KUKA KRL program: EPS_2_251825_SA34_A_20260116064118.src

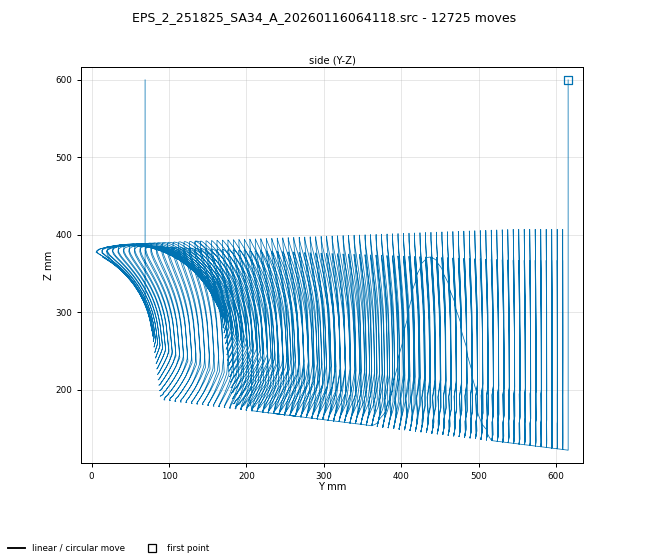
[picture p0: tool path of EPS_2_251825_SA34_A_20260116064118.src, 12725 of 12727 moves have a stored position in this frame; points joined in program order, loops and branches not executed]
&ACCESS RVP
&REL 4
&COMMENT QRS 19112012
&PARAM EDITMASK = *
DEF PART()
EXT BAS (BAS_COMMAND :IN,REAL :IN )
INT I
BAS (#INITMOV,0 )

;KUKA QRS Post kuka4.cps  Date:22-06-2017 !

File_ID=2990

QRS_PRE_INIT()

;Init var - Until changes are made in qrs_pre_init
Outlet_Square_prg=0
Inlet_1_Square_prg=0
Inlet_2_Square_prg=0
Inlet_3_Square_prg=0
Inlet_4_Square_prg=0
Inlet_5_Square_prg=0

Outlet_1={X 0.000, Y 546.330, Z 306.500, B 0.000, E1 0.000 }
Inlet_1={X 0.000, Y 549.180, Z 266.500, B 0.000, E1 160.000 }
Outlet_1_type=201
Inlet_1_type=201
;QRS#1=Sidecore dimensions
;QRS#2=200-8" PVC SDR 35
;QRS#3=200-8" PVC SDR 35
;QRS#4=
;QRS#5=
;QRS#6=
;QRS#7=
;QRS#8=
;QRS#9=12-08 PSX
;QRS#10=12-08 PSX
;QRS#11=
;QRS#12=
;QRS#13=
;QRS#14=
;QRS#15=
;QRS#16=1220x127x686 2,25'
;QRS#17=EPS Height
;QRS#18=407
;QRS#19=*
;QRS#20= UPDATED VERSION 22-06-2017
;QRS#21=*
Outlet_Square=0100
Inlet_1_Square=0100
Inlet_2_Square=0
Inlet_3_Square=0
Inlet_4_Square=0
Inlet_5_Square=0
Mill_Square=1
Outlet_Square_Prg=204
Inlet_1_Square_prg=204

QRS_INIT()

$ADVANCE=5

; T1
PTP {E1 173.645,E2 173.645}
PTP {X 0,Y 615.452,A -85,B 0,C 180,E1 173.645,E2 173.645,E3 0,E4 0,E5 0,E6 0}
QRS_SPEED_INIT()
LIN {X 0,Y 615.452,Z 600,A -85,B 0,C 180,E1 173.645,E2 173.645,E3 0,E4 0,E5 0,E6 0} C_VEL
LIN {X 0,Y 615.452,Z 131.871,A -85,B 0,C 180,E1 173.645,E2 173.645} C_VEL
LIN {X 0,Y 615.452,Z 123.693,A -85,B 0,C 180,E1 173.645,E2 173.645} C_VEL
LIN {X 0,Y 615.446,Z 121.693,A -85,B 0,C 180,E1 173.459,E2 173.459} C_VEL
LIN {X 0,Y 615.481,Z 121.699,A -85,B 0,C 180,E1 170.802,E2 170.802} C_VEL
LIN {X 0,Y 615.48,Z 121.688,A -85,B 0,C 180,E1 168.139,E2 168.139} C_VEL
LIN {X 0,Y 615.452,Z 121.694,A -85,B 0,C 180,E1 165.45,E2 165.45} C_VEL
LIN {X 0,Y 615.493,Z 121.695,A -85,B 0,C 180,E1 162.73,E2 162.73} C_VEL
LIN {X 0,Y 615.459,Z 121.69,A -85,B 0,C 180,E1 159.967,E2 159.967} C_VEL
LIN {X 0,Y 615.457,Z 121.693,A -85,B 0,C 180,E1 157.662,E2 157.662} C_VEL
LIN {X 0,Y 615.494,Z 121.696,A -85,B 0,C 180,E1 155.009,E2 155.009} C_VEL
LIN {X 0,Y 615.461,Z 121.69,A -85,B 0,C 180,E1 152.084,E2 152.084} C_VEL
LIN {X 0,Y 615.46,Z 121.694,A -85,B 0,C 180,E1 149.839,E2 149.839} C_VEL
LIN {X 0,Y 615.481,Z 121.699,A -85,B 0,C 180,E1 147.543,E2 147.543} C_VEL
LIN {X 0,Y 615.489,Z 121.693,A -85,B 0,C 180,E1 145.186,E2 145.186} C_VEL
LIN {X 0,Y 615.491,Z 121.683,A -85,B 0,C 180,E1 142.759,E2 142.759} C_VEL
LIN {X 0,Y 615.475,Z 121.697,A -85,B 0,C 180,E1 139.913,E2 139.913} C_VEL
LIN {X 0,Y 615.488,Z 121.684,A -85,B 0,C 180,E1 136.953,E2 136.953} C_VEL
LIN {X 0,Y 615.475,Z 121.695,A -85,B 0,C 180,E1 134.151,E2 134.151} C_VEL
LIN {X 0,Y 615.484,Z 121.69,A -85,B 0,C 180,E1 131.474,E2 131.474} C_VEL
LIN {X 0,Y 615.473,Z 121.689,A -85,B 0,C 180,E1 128.643,E2 128.643} C_VEL
LIN {X 0,Y 615.494,Z 136.384,A -85,B 0,C 180,E1 126.128,E2 126.128} C_VEL
LIN {X 0,Y 615.488,Z 153.64,A -85,B 0,C 180,E1 123.236,E2 123.236} C_VEL
LIN {X 0,Y 615.488,Z 156.2,A -85,B 0,C 180,E1 122.81,E2 122.81} C_VEL
LIN {X 0,Y 615.474,Z 263.278,A -85,B 0,C 180,E1 121.536,E2 121.536} C_VEL
LIN {X 0,Y 615.497,Z 276.678,A -85,B 0,C 180,E1 121.236,E2 121.236} C_VEL
LIN {X 0,Y 615.493,Z 289.09,A -85,B 0,C 180,E1 120.824,E2 120.824} C_VEL
LIN {X 0,Y 615.469,Z 299.786,A -85,B 0,C 180,E1 120.351,E2 120.351} C_VEL
LIN {X 0,Y 615.47,Z 311.326,A -85,B 0,C 180,E1 119.695,E2 119.695} C_VEL
LIN {X 0,Y 615.499,Z 321.929,A -85,B 0,C 180,E1 118.938,E2 118.938} C_VEL
LIN {X 0,Y 615.497,Z 330.569,A -85,B 0,C 180,E1 118.184,E2 118.184} C_VEL
LIN {X 0,Y 615.498,Z 338.385,A -85,B 0,C 180,E1 117.361,E2 117.361} C_VEL
LIN {X 0,Y 615.494,Z 345.548,A -85,B 0,C 180,E1 116.444,E2 116.444} C_VEL
LIN {X 0,Y 615.495,Z 352.739,A -85,B 0,C 180,E1 115.281,E2 115.281} C_VEL
LIN {X 0,Y 615.496,Z 357.591,A -85,B 0,C 180,E1 114.272,E2 114.272} C_VEL
LIN {X 0,Y 615.495,Z 361.489,A -85,B 0,C 180,E1 113.2,E2 113.2} C_VEL
LIN {X 0,Y 615.497,Z 364.191,A -85,B 0,C 180,E1 112.136,E2 112.136} C_VEL
LIN {X 0,Y 615.498,Z 365.382,A -85,B 0,C 180,E1 111.432,E2 111.432} C_VEL
LIN {X 0,Y 615.495,Z 366.208,A -85,B 0,C 180,E1 110.56,E2 110.56} C_VEL
LIN {X 0,Y 615.496,Z 366.2,A -85,B 0,C 180,E1 109.338,E2 109.338} C_VEL
LIN {X 0,Y 615.495,Z 365.535,A -85,B 0,C 180,E1 108.608,E2 108.608} C_VEL
LIN {X 0,Y 615.497,Z 364.55,A -85,B 0,C 180,E1 107.957,E2 107.957} C_VEL
LIN {X 0,Y 615.495,Z 363.056,A -85,B 0,C 180,E1 107.27,E2 107.27} C_VEL
LIN {X 0,Y 615.495,Z 360.608,A -85,B 0,C 180,E1 106.435,E2 106.435} C_VEL
LIN {X 0,Y 615.497,Z 355.768,A -85,B 0,C 180,E1 105.226,E2 105.226} C_VEL
LIN {X 0,Y 615.495,Z 350.565,A -85,B 0,C 180,E1 104.244,E2 104.244} C_VEL
LIN {X 0,Y 615.497,Z 343.595,A -85,B 0,C 180,E1 103.201,E2 103.201} C_VEL
LIN {X 0,Y 615.497,Z 335.207,A -85,B 0,C 180,E1 102.195,E2 102.195} C_VEL
LIN {X 0,Y 615.499,Z 326.571,A -85,B 0,C 180,E1 101.36,E2 101.36} C_VEL
LIN {X 0,Y 615.494,Z 315.975,A -85,B 0,C 180,E1 100.527,E2 100.527} C_VEL
LIN {X 0,Y 615.495,Z 305.473,A -85,B 0,C 180,E1 99.862,E2 99.862} C_VEL
LIN {X 0,Y 615.497,Z 293.798,A -85,B 0,C 180,E1 99.281,E2 99.281} C_VEL
LIN {X 0,Y 615.462,Z 281.785,A -85,B 0,C 180,E1 98.826,E2 98.826} C_VEL
LIN {X 0,Y 615.454,Z 269.574,A -85,B 0,C 180,E1 98.496,E2 98.496} C_VEL
LIN {X 0,Y 615.459,Z 257.497,A -85,B 0,C 180,E1 98.289,E2 98.289} C_VEL
LIN {X 0,Y 615.464,Z 156.157,A -85,B 0,C 180,E1 97.092,E2 97.092} C_VEL
LIN {X 0,Y 615.44,Z 141.171,A -85,B 0,C 180,E1 94.585,E2 94.585} C_VEL
LIN {X 0,Y 615.499,Z 125.645,A -85,B 0,C 180,E1 91.963,E2 91.963} C_VEL
LIN {X 0,Y 615.429,Z 121.699,A -85,B 0,C 180,E1 91.268,E2 91.268} C_VEL
LIN {X 0,Y 615.43,Z 121.699,A -85,B 0,C 180,E1 89.346,E2 89.346} C_VEL
LIN {X 0,Y 615.429,Z 121.699,A -85,B 0,C 180,E1 87.382,E2 87.382} C_VEL
LIN {X 0,Y 615.427,Z 121.699,A -85,B 0,C 180,E1 85.415,E2 85.415} C_VEL
LIN {X 0,Y 615.427,Z 121.699,A -85,B 0,C 180,E1 83.443,E2 83.443} C_VEL
LIN {X 0,Y 615.425,Z 121.699,A -85,B 0,C 180,E1 81.462,E2 81.462} C_VEL
LIN {X 0,Y 615.416,Z 121.699,A -85,B 0,C 180,E1 79.144,E2 79.144} C_VEL
LIN {X 0,Y 615.435,Z 121.699,A -85,B 0,C 180,E1 76.797,E2 76.797} C_VEL
LIN {X 0,Y 615.466,Z 121.7,A -85,B 0,C 180,E1 74.094,E2 74.094} C_VEL
LIN {X 0,Y 615.414,Z 121.699,A -85,B 0,C 180,E1 71.351,E2 71.351} C_VEL
LIN {X 0,Y 615.485,Z 121.699,A -85,B 0,C 180,E1 68.568,E2 68.568} C_VEL
LIN {X 0,Y 615.416,Z 121.7,A -85,B 0,C 180,E1 65.725,E2 65.725} C_VEL
LIN {X 0,Y 615.41,Z 121.7,A -85,B 0,C 180,E1 63.552,E2 63.552} C_VEL
LIN {X 0,Y 615.477,Z 121.703,A -85,B 0,C 180,E1 60.593,E2 60.593} C_VEL
LIN {X 0,Y 615.445,Z 121.7,A -85,B 0,C 180,E1 58.312,E2 58.312} C_VEL
LIN {X 0,Y 615.416,Z 121.7,A -85,B 0,C 180,E1 55.973,E2 55.973} C_VEL
LIN {X 0,Y 615.464,Z 121.7,A -85,B 0,C 180,E1 53.066,E2 53.066} C_VEL
LIN {X 0,Y 615.422,Z 121.7,A -85,B 0,C 180,E1 50.244,E2 50.244} C_VEL
LIN {X 0,Y 615.414,Z 121.699,A -85,B 0,C 180,E1 47.927,E2 47.927} C_VEL
LIN {X 0,Y 615.416,Z 121.7,A -85,B 0,C 180,E1 45.843,E2 45.843} C_VEL
LIN {X 0,Y 615.475,Z 121.7,A -85,B 0,C 180,E1 43.245,E2 43.245} C_VEL
LIN {X 0,Y 615.437,Z 121.698,A -85,B 0,C 180,E1 40.61,E2 40.61} C_VEL
LIN {X 0,Y 615.466,Z 121.698,A -85,B 0,C 180,E1 38.905,E2 38.905} C_VEL
LIN {X 0,Y 615.421,Z 121.699,A -85,B 0,C 180,E1 36.429,E2 36.429} C_VEL
LIN {X 0,Y 615.469,Z 121.7,A -85,B 0,C 180,E1 33.531,E2 33.531} C_VEL
LIN {X 0,Y 615.447,Z 121.698,A -85,B 0,C 180,E1 30.921,E2 30.921} C_VEL
LIN {X 0,Y 615.419,Z 121.698,A -85,B 0,C 180,E1 28.437,E2 28.437} C_VEL
LIN {X 0,Y 615.471,Z 121.7,A -85,B 0,C 180,E1 25.716,E2 25.716} C_VEL
LIN {X 0,Y 615.428,Z 121.697,A -85,B 0,C 180,E1 22.846,E2 22.846} C_VEL
LIN {X 0,Y 615.421,Z 121.698,A -85,B 0,C 180,E1 20.539,E2 20.539} C_VEL
LIN {X 0,Y 615.465,Z 121.699,A -85,B 0,C 180,E1 17.957,E2 17.957} C_VEL
LIN {X 0,Y 615.445,Z 121.696,A -85,B 0,C 180,E1 15.227,E2 15.227} C_VEL
LIN {X 0,Y 615.439,Z 121.697,A -85,B 0,C 180,E1 13.202,E2 13.202} C_VEL
LIN {X 0,Y 615.423,Z 121.697,A -85,B 0,C 180,E1 10.854,E2 10.854} C_VEL
LIN {X 0,Y 615.434,Z 121.698,A -85,B 0,C 180,E1 8.537,E2 8.537} C_VEL
LIN {X 0,Y 615.499,Z 121.696,A -85,B 0,C 180,E1 5.898,E2 5.898} C_VEL
LIN {X 0,Y 615.431,Z 121.696,A -85,B 0,C 180,E1 3.273,E2 3.273} C_VEL
LIN {X 0,Y 615.429,Z 121.697,A -85,B 0,C 180,E1 1.308,E2 1.308} C_VEL
LIN {X 0,Y 615.431,Z 121.696,A -85,B 0,C 180,E1 -0.655,E2 -0.655} C_VEL
LIN {X 0,Y 615.429,Z 121.697,A -85,B 0,C 180,E1 -2.618,E2 -2.618} C_VEL
LIN {X 0,Y 615.431,Z 121.696,A -85,B 0,C 180,E1 -4.585,E2 -4.585} C_VEL
LIN {X 0,Y 615.431,Z 121.696,A -85,B 0,C 180,E1 -6.558,E2 -6.558} C_VEL
LIN {X 0,Y 615.43,Z 121.696,A -85,B 0,C 180,E1 -8.538,E2 -8.538} C_VEL
LIN {X 0,Y 615.431,Z 121.697,A -85,B 0,C 180,E1 -10.858,E2 -10.858} C_VEL
LIN {X 0,Y 615.456,Z 121.7,A -85,B 0,C 180,E1 -13.202,E2 -13.202} C_VEL
LIN {X 0,Y 615.465,Z 121.694,A -85,B 0,C 180,E1 -15.906,E2 -15.906} C_VEL
LIN {X 0,Y 615.454,Z 121.694,A -85,B 0,C 180,E1 -17.958,E2 -17.958} C_VEL
LIN {X 0,Y 615.431,Z 121.697,A -85,B 0,C 180,E1 -20.541,E2 -20.541} C_VEL
LIN {X 0,Y 615.45,Z 121.698,A -85,B 0,C 180,E1 -22.846,E2 -22.846} C_VEL
LIN {X 0,Y 615.463,Z 121.693,A -85,B 0,C 180,E1 -25.717,E2 -25.717} C_VEL
LIN {X 0,Y 615.441,Z 121.694,A -85,B 0,C 180,E1 -27.918,E2 -27.918} C_VEL
LIN {X 0,Y 615.432,Z 121.695,A -85,B 0,C 180,E1 -30.163,E2 -30.163} C_VEL
LIN {X 0,Y 615.441,Z 121.697,A -85,B 0,C 180,E1 -32.461,E2 -32.461} C_VEL
LIN {X 0,Y 615.478,Z 121.7,A -85,B 0,C 180,E1 -34.816,E2 -34.816} C_VEL
LIN {X 0,Y 615.487,Z 121.692,A -85,B 0,C 180,E1 -37.243,E2 -37.243} C_VEL
LIN {X 0,Y 615.436,Z 121.695,A -85,B 0,C 180,E1 -39.754,E2 -39.754} C_VEL
LIN {X 0,Y 615.434,Z 121.697,A -85,B 0,C 180,E1 -42.074,E2 -42.074} C_VEL
LIN {X 0,Y 615.442,Z 121.697,A -85,B 0,C 180,E1 -44.154,E2 -44.154} C_VEL
LIN {X 0,Y 615.488,Z 121.693,A -85,B 0,C 180,E1 -46.953,E2 -46.953} C_VEL
LIN {X 0,Y 615.448,Z 121.693,A -85,B 0,C 180,E1 -49.39,E2 -49.39} C_VEL
LIN {X 0,Y 615.445,Z 121.697,A -85,B 0,C 180,E1 -51.994,E2 -51.994} C_VEL
LIN {X 0,Y 615.487,Z 121.699,A -85,B 0,C 180,E1 -54.384,E2 -54.384} C_VEL
LIN {X 0,Y 615.486,Z 121.692,A -85,B 0,C 180,E1 -56.763,E2 -56.763} C_VEL
LIN {X 0,Y 615.456,Z 121.692,A -85,B 0,C 180,E1 -59.078,E2 -59.078} C_VEL
LIN {X 0,Y 615.439,Z 121.695,A -85,B 0,C 180,E1 -61.559,E2 -61.559} C_VEL
LIN {X 0,Y 615.494,Z 121.694,A -85,B 0,C 180,E1 -64.431,E2 -64.431} C_VEL
LIN {X 0,Y 615.442,Z 121.693,A -85,B 0,C 180,E1 -67.153,E2 -67.153} C_VEL
LIN {X 0,Y 615.441,Z 121.787,A -85,B 0,C 180,E1 -67.44,E2 -67.44} C_VEL
LIN {X 0,Y 615.478,Z 140.396,A -85,B 0,C 180,E1 -69.967,E2 -69.967} C_VEL
LIN {X 0,Y 615.47,Z 161.075,A -85,B 0,C 180,E1 -72.729,E2 -72.729} C_VEL
LIN {X 0,Y 615.472,Z 181.731,A -85,B 0,C 180,E1 -75.45,E2 -75.45} C_VEL
LIN {X 0,Y 615.454,Z 194.469,A -85,B 0,C 180,E1 -77.113,E2 -77.113} C_VEL
LIN {X 0,Y 615.488,Z 302.818,A -85,B 0,C 180,E1 -78.41,E2 -78.41} C_VEL
LIN {X 0,Y 615.477,Z 315.338,A -85,B 0,C 180,E1 -78.681,E2 -78.681} C_VEL
LIN {X 0,Y 615.488,Z 328.619,A -85,B 0,C 180,E1 -79.113,E2 -79.113} C_VEL
LIN {X 0,Y 615.477,Z 340.475,A -85,B 0,C 180,E1 -79.639,E2 -79.639} C_VEL
LIN {X 0,Y 615.494,Z 351.991,A -85,B 0,C 180,E1 -80.304,E2 -80.304} C_VEL
LIN {X 0,Y 615.499,Z 362.339,A -85,B 0,C 180,E1 -81.05,E2 -81.05} C_VEL
LIN {X 0,Y 615.497,Z 370.81,A -85,B 0,C 180,E1 -81.794,E2 -81.794} C_VEL
LIN {X 0,Y 615.498,Z 378.605,A -85,B 0,C 180,E1 -82.619,E2 -82.619} C_VEL
LIN {X 0,Y 615.496,Z 386.202,A -85,B 0,C 180,E1 -83.608,E2 -83.608} C_VEL
LIN {X 0,Y 615.498,Z 393.204,A -85,B 0,C 180,E1 -84.759,E2 -84.759} C_VEL
LIN {X 0,Y 615.494,Z 397.851,A -85,B 0,C 180,E1 -85.743,E2 -85.743} C_VEL
LIN {X 0,Y 615.494,Z 401.398,A -85,B 0,C 180,E1 -86.727,E2 -86.727} C_VEL
LIN {X 0,Y 615.497,Z 403.233,A -85,B 0,C 180,E1 -87.382,E2 -87.382} C_VEL
LIN {X 0,Y 615.5,Z 404.607,A -85,B 0,C 180,E1 -88.037,E2 -88.037} C_VEL
LIN {X 0,Y 615.496,Z 406.173,A -85,B 0,C 180,E1 -89.346,E2 -89.346} C_VEL
LIN {X 0,Y 615.494,Z 406.389,A -85,B 0,C 180,E1 -90,E2 -90} C_VEL
LIN {X 0,Y 615.495,Z 405.58,A -85,B 0,C 180,E1 -91.308,E2 -91.308} C_VEL
LIN {X 0,Y 615.5,Z 404.608,A -85,B 0,C 180,E1 -91.963,E2 -91.963} C_VEL
LIN {X 0,Y 615.497,Z 403.233,A -85,B 0,C 180,E1 -92.618,E2 -92.618} C_VEL
LIN {X 0,Y 615.496,Z 400.35,A -85,B 0,C 180,E1 -93.601,E2 -93.601} C_VEL
LIN {X 0,Y 615.498,Z 396.442,A -85,B 0,C 180,E1 -94.584,E2 -94.584} C_VEL
LIN {X 0,Y 615.499,Z 391.405,A -85,B 0,C 180,E1 -95.57,E2 -95.57} C_VEL
LIN {X 0,Y 615.497,Z 384.87,A -85,B 0,C 180,E1 -96.583,E2 -96.583} C_VEL
LIN {X 0,Y 615.497,Z 377.134,A -85,B 0,C 180,E1 -97.545,E2 -97.545} C_VEL
LIN {X 0,Y 615.498,Z 369.045,A -85,B 0,C 180,E1 -98.371,E2 -98.371} C_VEL
LIN {X 0,Y 615.499,Z 359.168,A -85,B 0,C 180,E1 -99.199,E2 -99.199} C_VEL
LIN {X 0,Y 615.488,Z 347.982,A -85,B 0,C 180,E1 -99.945,E2 -99.945} C_VEL
LIN {X 0,Y 615.482,Z 337.024,A -85,B 0,C 180,E1 -100.527,E2 -100.527} C_VEL
LIN {X 0,Y 615.48,Z 324.491,A -85,B 0,C 180,E1 -101.04,E2 -101.04} C_VEL
LIN {X 0,Y 615.479,Z 312.068,A -85,B 0,C 180,E1 -101.402,E2 -101.402} C_VEL
LIN {X 0,Y 615.493,Z 298.466,A -85,B 0,C 180,E1 -101.652,E2 -101.652} C_VEL
LIN {X 0,Y 615.454,Z 194.471,A -85,B 0,C 180,E1 -102.887,E2 -102.887} C_VEL
LIN {X 0,Y 615.496,Z 172.696,A -85,B 0,C 180,E1 -105.735,E2 -105.735} C_VEL
LIN {X 0,Y 615.455,Z 152.319,A -85,B 0,C 180,E1 -108.436,E2 -108.436} C_VEL
LIN {X 0,Y 615.475,Z 132.637,A -85,B 0,C 180,E1 -111.081,E2 -111.081} C_VEL
LIN {X 0,Y 615.44,Z 121.695,A -85,B 0,C 180,E1 -112.592,E2 -112.592} C_VEL
LIN {X 0,Y 615.451,Z 121.692,A -85,B 0,C 180,E1 -114.993,E2 -114.993} C_VEL
LIN {X 0,Y 615.468,Z 121.699,A -85,B 0,C 180,E1 -117.916,E2 -117.916} C_VEL
LIN {X 0,Y 615.442,Z 121.697,A -85,B 0,C 180,E1 -120.163,E2 -120.163} C_VEL
LIN {X 0,Y 615.432,Z 121.696,A -85,B 0,C 180,E1 -122.461,E2 -122.461} C_VEL
LIN {X 0,Y 615.451,Z 121.694,A -85,B 0,C 180,E1 -124.818,E2 -124.818} C_VEL
LIN {X 0,Y 615.495,Z 121.697,A -85,B 0,C 180,E1 -127.242,E2 -127.242} C_VEL
LIN {X 0,Y 615.444,Z 121.699,A -85,B 0,C 180,E1 -129.754,E2 -129.754} C_VEL
LIN {X 0,Y 615.425,Z 121.698,A -85,B 0,C 180,E1 -132.073,E2 -132.073} C_VEL
LIN {X 0,Y 615.423,Z 121.698,A -85,B 0,C 180,E1 -134.156,E2 -134.156} C_VEL
LIN {X 0,Y 615.469,Z 121.697,A -85,B 0,C 180,E1 -136.753,E2 -136.753} C_VEL
LIN {X 0,Y 615.444,Z 121.7,A -85,B 0,C 180,E1 -139.39,E2 -139.39} C_VEL
LIN {X 0,Y 615.473,Z 121.7,A -85,B 0,C 180,E1 -141.094,E2 -141.094} C_VEL
LIN {X 0,Y 615.418,Z 121.7,A -85,B 0,C 180,E1 -143.57,E2 -143.57} C_VEL
LIN {X 0,Y 615.46,Z 121.7,A -85,B 0,C 180,E1 -146.47,E2 -146.47} C_VEL
LIN {X 0,Y 615.446,Z 121.699,A -85,B 0,C 180,E1 -149.078,E2 -149.078} C_VEL
LIN {X 0,Y 615.417,Z 121.699,A -85,B 0,C 180,E1 -151.562,E2 -151.562} C_VEL
LIN {X 0,Y 615.47,Z 121.7,A -85,B 0,C 180,E1 -154.283,E2 -154.283} C_VEL
LIN {X 0,Y 615.43,Z 121.697,A -85,B 0,C 180,E1 -157.153,E2 -157.153} C_VEL
LIN {X 0,Y 615.424,Z 121.698,A -85,B 0,C 180,E1 -159.46,E2 -159.46} C_VEL
LIN {X 0,Y 615.473,Z 121.699,A -85,B 0,C 180,E1 -162.042,E2 -162.042} C_VEL
LIN {X 0,Y 615.448,Z 121.695,A -85,B 0,C 180,E1 -164.773,E2 -164.773} C_VEL
LIN {X 0,Y 615.443,Z 121.695,A -85,B 0,C 180,E1 -166.797,E2 -166.797} C_VEL
LIN {X 0,Y 615.432,Z 121.696,A -85,B 0,C 180,E1 -169.141,E2 -169.141} C_VEL
LIN {X 0,Y 615.448,Z 121.698,A -85,B 0,C 180,E1 -171.462,E2 -171.462} C_VEL
LIN {X 0,Y 615.499,Z 121.691,A -85,B 0,C 180,E1 -174.101,E2 -174.101} C_VEL
LIN {X 0,Y 615.44,Z 121.694,A -85,B 0,C 180,E1 -176.726,E2 -176.726} C_VEL
LIN {X 0,Y 615.441,Z 121.694,A -85,B 0,C 180,E1 -178.691,E2 -178.691} C_VEL
LIN {X 0,Y 615.465,Z 121.698,A -85,B 0,C 180,E1 -181.308,E2 -181.308} C_VEL
LIN {X 0,Y 615.486,Z 121.691,A -85,B 0,C 180,E1 -183.928,E2 -183.928} C_VEL
LIN {X 0,Y 615.446,Z 121.693,A -85,B 0,C 180,E1 -186.541,E2 -186.541} C_VEL
LIN {X 0,Y 614.789,Z 121.846,A -85,B 0,C 180,E1 -187.087,E2 -187.087} C_VEL
LIN {X 0,Y 611.974,Z 122.251,A -85,B 0,C 180,E1 -187.974,E2 -187.974} C_VEL
LIN {X 0,Y 609.586,Z 122.567,A -85,B 0,C 180,E1 -188.686,E2 -188.686} C_VEL
LIN {X 0,Y 608.549,Z 122.687,A -85,B 0,C 180,E1 -189.236,E2 -189.236} C_VEL
LIN {X 0,Y 608.459,Z 122.695,A -85,B 0,C 180,E1 -189.422,E2 -189.422} C_VEL
LIN {X 0,Y 608.451,Z 122.689,A -85,B 0,C 180,E1 -192,E2 -192} C_VEL
LIN {X 0,Y 608.449,Z 122.688,A -85,B 0,C 180,E1 -194.038,E2 -194.038} C_VEL
LIN {X 0,Y 608.45,Z 122.69,A -85,B 0,C 180,E1 -196.522,E2 -196.522} C_VEL
LIN {X 0,Y 608.448,Z 122.69,A -85,B 0,C 180,E1 -199.57,E2 -199.57} C_VEL
LIN {X 0,Y 608.434,Z 122.692,A -85,B 0,C 180,E1 -202.406,E2 -202.406} C_VEL
LIN {X 0,Y 608.453,Z 122.691,A -85,B 0,C 180,E1 -205.3,E2 -205.3} C_VEL
LIN {X 0,Y 608.442,Z 122.69,A -85,B 0,C 180,E1 -207.518,E2 -207.518} C_VEL
LIN {X 0,Y 608.446,Z 122.689,A -85,B 0,C 180,E1 -209.967,E2 -209.967} C_VEL
LIN {X 0,Y 608.457,Z 122.693,A -85,B 0,C 180,E1 -212.879,E2 -212.879} C_VEL
LIN {X 0,Y 608.435,Z 122.691,A -85,B 0,C 180,E1 -215.278,E2 -215.278} C_VEL
LIN {X 0,Y 608.461,Z 122.688,A -85,B 0,C 180,E1 -217.746,E2 -217.746} C_VEL
LIN {X 0,Y 608.447,Z 122.699,A -85,B 0,C 180,E1 -220.328,E2 -220.328} C_VEL
LIN {X 0,Y 608.456,Z 122.688,A -85,B 0,C 180,E1 -222.959,E2 -222.959} C_VEL
LIN {X 0,Y 608.447,Z 122.692,A -85,B 0,C 180,E1 -225.736,E2 -225.736} C_VEL
LIN {X 0,Y 608.462,Z 122.689,A -85,B 0,C 180,E1 -228.657,E2 -228.657} C_VEL
LIN {X 0,Y 608.462,Z 122.787,A -85,B 0,C 180,E1 -231.332,E2 -231.332} C_VEL
LIN {X 0,Y 608.479,Z 138.082,A -85,B 0,C 180,E1 -233.95,E2 -233.95} C_VEL
LIN {X 0,Y 608.46,Z 154.529,A -85,B 0,C 180,E1 -236.726,E2 -236.726} C_VEL
LIN {X 0,Y 608.473,Z 156.462,A -85,B 0,C 180,E1 -237.044,E2 -237.044} C_VEL
LIN {X 0,Y 608.534,Z 263.716,A -85,B 0,C 180,E1 -238.336,E2 -238.336} C_VEL
LIN {X 0,Y 608.534,Z 277.004,A -85,B 0,C 180,E1 -238.639,E2 -238.639} C_VEL
LIN {X 0,Y 608.526,Z 289.836,A -85,B 0,C 180,E1 -239.073,E2 -239.073} C_VEL
LIN {X 0,Y 608.486,Z 301.644,A -85,B 0,C 180,E1 -239.618,E2 -239.618} C_VEL
LIN {X 0,Y 608.463,Z 313.409,A -85,B 0,C 180,E1 -240.315,E2 -240.315} C_VEL
LIN {X 0,Y 608.488,Z 323.927,A -85,B 0,C 180,E1 -241.098,E2 -241.098} C_VEL
LIN {X 0,Y 608.485,Z 332.9,A -85,B 0,C 180,E1 -241.923,E2 -241.923} C_VEL
LIN {X 0,Y 608.462,Z 341.754,A -85,B 0,C 180,E1 -242.92,E2 -242.92} C_VEL
LIN {X 0,Y 608.434,Z 349.174,A -85,B 0,C 180,E1 -243.964,E2 -243.964} C_VEL
LIN {X 0,Y 608.43,Z 355.309,A -85,B 0,C 180,E1 -245.063,E2 -245.063} C_VEL
LIN {X 0,Y 608.441,Z 359.985,A -85,B 0,C 180,E1 -246.154,E2 -246.154} C_VEL
LIN {X 0,Y 608.44,Z 362.405,A -85,B 0,C 180,E1 -246.876,E2 -246.876} C_VEL
LIN {X 0,Y 608.429,Z 364.248,A -85,B 0,C 180,E1 -247.593,E2 -247.593} C_VEL
LIN {X 0,Y 608.419,Z 365.612,A -85,B 0,C 180,E1 -248.307,E2 -248.307} C_VEL
LIN {X 0,Y 608.44,Z 366.744,A -85,B 0,C 180,E1 -249.327,E2 -249.327} C_VEL
LIN {X 0,Y 608.416,Z 366.916,A -85,B 0,C 180,E1 -250.428,E2 -250.428} C_VEL
LIN {X 0,Y 608.426,Z 366.271,A -85,B 0,C 180,E1 -251.295,E2 -251.295} C_VEL
LIN {X 0,Y 608.419,Z 364.193,A -85,B 0,C 180,E1 -252.522,E2 -252.522} C_VEL
LIN {X 0,Y 608.426,Z 361.552,A -85,B 0,C 180,E1 -253.483,E2 -253.483} C_VEL
LIN {X 0,Y 608.43,Z 357.335,A -85,B 0,C 180,E1 -254.593,E2 -254.593} C_VEL
LIN {X 0,Y 608.434,Z 352.189,A -85,B 0,C 180,E1 -255.62,E2 -255.62} C_VEL
LIN {X 0,Y 608.445,Z 345.722,A -85,B 0,C 180,E1 -256.643,E2 -256.643} C_VEL
LIN {X 0,Y 608.46,Z 337.624,A -85,B 0,C 180,E1 -257.662,E2 -257.662} C_VEL
LIN {X 0,Y 608.469,Z 329.402,A -85,B 0,C 180,E1 -258.507,E2 -258.507} C_VEL
LIN {X 0,Y 608.5,Z 319.397,A -85,B 0,C 180,E1 -259.351,E2 -259.351} C_VEL
LIN {X 0,Y 608.492,Z 308.141,A -85,B 0,C 180,E1 -260.107,E2 -260.107} C_VEL
LIN {X 0,Y 608.51,Z 297.156,A -85,B 0,C 180,E1 -260.695,E2 -260.695} C_VEL
LIN {X 0,Y 608.511,Z 285.043,A -85,B 0,C 180,E1 -261.197,E2 -261.197} C_VEL
LIN {X 0,Y 608.521,Z 272.391,A -85,B 0,C 180,E1 -261.574,E2 -261.574} C_VEL
LIN {X 0,Y 608.511,Z 259.154,A -85,B 0,C 180,E1 -261.825,E2 -261.825} C_VEL
LIN {X 0,Y 608.45,Z 156.374,A -85,B 0,C 180,E1 -263.055,E2 -263.055} C_VEL
LIN {X 0,Y 608.441,Z 140.716,A -85,B 0,C 180,E1 -265.694,E2 -265.694} C_VEL
LIN {X 0,Y 608.444,Z 123.264,A -85,B 0,C 180,E1 -268.676,E2 -268.676} C_VEL
LIN {X 0,Y 608.413,Z 122.694,A -85,B 0,C 180,E1 -268.8,E2 -268.8} C_VEL
LIN {X 0,Y 608.408,Z 122.695,A -85,B 0,C 180,E1 -270.662,E2 -270.662} C_VEL
LIN {X 0,Y 608.425,Z 122.693,A -85,B 0,C 180,E1 -272.648,E2 -272.648} C_VEL
LIN {X 0,Y 608.413,Z 122.694,A -85,B 0,C 180,E1 -275.302,E2 -275.302} C_VEL
LIN {X 0,Y 608.464,Z 122.695,A -85,B 0,C 180,E1 -277.967,E2 -277.967} C_VEL
LIN {X 0,Y 608.402,Z 122.694,A -85,B 0,C 180,E1 -280.651,E2 -280.651} C_VEL
LIN {X 0,Y 608.425,Z 122.695,A -85,B 0,C 180,E1 -283.358,E2 -283.358} C_VEL
LIN {X 0,Y 608.425,Z 122.695,A -85,B 0,C 180,E1 -286.095,E2 -286.095} C_VEL
LIN {X 0,Y 608.396,Z 122.695,A -85,B 0,C 180,E1 -288.872,E2 -288.872} C_VEL
LIN {X 0,Y 608.447,Z 122.696,A -85,B 0,C 180,E1 -291.693,E2 -291.693} C_VEL
LIN {X 0,Y 608.402,Z 122.694,A -85,B 0,C 180,E1 -294.574,E2 -294.574} C_VEL
LIN {X 0,Y 608.456,Z 122.694,A -85,B 0,C 180,E1 -297.204,E2 -297.204} C_VEL
LIN {X 0,Y 608.4,Z 122.696,A -85,B 0,C 180,E1 -299.961,E2 -299.961} C_VEL
LIN {X 0,Y 608.402,Z 122.694,A -85,B 0,C 180,E1 -302.514,E2 -302.514} C_VEL
LIN {X 0,Y 608.406,Z 122.703,A -85,B 0,C 180,E1 -305.281,E2 -305.281} C_VEL
LIN {X 0,Y 608.423,Z 122.693,A -85,B 0,C 180,E1 -307.75,E2 -307.75} C_VEL
LIN {X 0,Y 608.4,Z 122.695,A -85,B 0,C 180,E1 -310.324,E2 -310.324} C_VEL
LIN {X 0,Y 608.439,Z 122.699,A -85,B 0,C 180,E1 -312.962,E2 -312.962} C_VEL
LIN {X 0,Y 608.4,Z 122.695,A -85,B 0,C 180,E1 -315.742,E2 -315.742} C_VEL
LIN {X 0,Y 608.401,Z 122.694,A -85,B 0,C 180,E1 -317.934,E2 -317.934} C_VEL
LIN {X 0,Y 608.433,Z 122.699,A -85,B 0,C 180,E1 -320.708,E2 -320.708} C_VEL
LIN {X 0,Y 608.432,Z 122.695,A -85,B 0,C 180,E1 -323.084,E2 -323.084} C_VEL
LIN {X 0,Y 608.42,Z 122.692,A -85,B 0,C 180,E1 -325.528,E2 -325.528} C_VEL
LIN {X 0,Y 608.416,Z 122.693,A -85,B 0,C 180,E1 -327.903,E2 -327.903} C_VEL
LIN {X 0,Y 608.435,Z 122.694,A -85,B 0,C 180,E1 -330.219,E2 -330.219} C_VEL
LIN {X 0,Y 608.398,Z 122.695,A -85,B 0,C 180,E1 -333.224,E2 -333.224} C_VEL
LIN {X 0,Y 608.409,Z 122.693,A -85,B 0,C 180,E1 -335.427,E2 -335.427} C_VEL
LIN {X 0,Y 608.451,Z 122.697,A -85,B 0,C 180,E1 -338.308,E2 -338.308} C_VEL
LIN {X 0,Y 608.411,Z 122.693,A -85,B 0,C 180,E1 -341.302,E2 -341.302} C_VEL
LIN {X 0,Y 608.432,Z 122.695,A -85,B 0,C 180,E1 -343.906,E2 -343.906} C_VEL
LIN {X 0,Y 608.432,Z 122.693,A -85,B 0,C 180,E1 -346.643,E2 -346.643} C_VEL
LIN {X 0,Y 608.41,Z 122.693,A -85,B 0,C 180,E1 -349.35,E2 -349.35} C_VEL
LIN {X 0,Y 608.472,Z 122.696,A -85,B 0,C 180,E1 -352.033,E2 -352.033} C_VEL
LIN {X 0,Y 608.418,Z 122.693,A -85,B 0,C 180,E1 -354.698,E2 -354.698} C_VEL
LIN {X 0,Y 608.434,Z 122.692,A -85,B 0,C 180,E1 -357.352,E2 -357.352} C_VEL
LIN {X 0,Y 608.478,Z 122.692,A -85,B 0,C 180,E1 -360,E2 -360} C_VEL
LIN {X 0,Y 608.426,Z 122.691,A -85,B 0,C 180,E1 -362.649,E2 -362.649} C_VEL
LIN {X 0,Y 608.431,Z 122.694,A -85,B 0,C 180,E1 -365.303,E2 -365.303} C_VEL
LIN {X 0,Y 608.469,Z 122.69,A -85,B 0,C 180,E1 -367.967,E2 -367.967} C_VEL
LIN {X 0,Y 608.432,Z 122.692,A -85,B 0,C 180,E1 -370.935,E2 -370.935} C_VEL
LIN {X 0,Y 608.44,Z 122.697,A -85,B 0,C 180,E1 -373.357,E2 -373.357} C_VEL
LIN {X 0,Y 608.429,Z 122.692,A -85,B 0,C 180,E1 -376.095,E2 -376.095} C_VEL
LIN {X 0,Y 608.436,Z 122.692,A -85,B 0,C 180,E1 -378.871,E2 -378.871} C_VEL
LIN {X 0,Y 608.458,Z 122.691,A -85,B 0,C 180,E1 -381.692,E2 -381.692} C_VEL
LIN {X 0,Y 608.422,Z 122.693,A -85,B 0,C 180,E1 -384.573,E2 -384.573} C_VEL
LIN {X 0,Y 608.482,Z 122.694,A -85,B 0,C 180,E1 -387.207,E2 -387.207} C_VEL
LIN {X 0,Y 608.412,Z 122.693,A -85,B 0,C 180,E1 -389.961,E2 -389.961} C_VEL
LIN {X 0,Y 608.425,Z 122.694,A -85,B 0,C 180,E1 -392.516,E2 -392.516} C_VEL
LIN {X 0,Y 608.423,Z 122.696,A -85,B 0,C 180,E1 -395.279,E2 -395.279} C_VEL
LIN {X 0,Y 608.437,Z 122.69,A -85,B 0,C 180,E1 -397.749,E2 -397.749} C_VEL
LIN {X 0,Y 608.438,Z 122.692,A -85,B 0,C 180,E1 -400.327,E2 -400.327} C_VEL
LIN {X 0,Y 608.461,Z 122.689,A -85,B 0,C 180,E1 -403.307,E2 -403.307} C_VEL
LIN {X 0,Y 608.435,Z 122.692,A -85,B 0,C 180,E1 -406.127,E2 -406.127} C_VEL
LIN {X 0,Y 608.457,Z 122.694,A -85,B 0,C 180,E1 -408.823,E2 -408.823} C_VEL
LIN {X 0,Y 608.416,Z 122.692,A -85,B 0,C 180,E1 -411.407,E2 -411.407} C_VEL
LIN {X 0,Y 608.437,Z 122.692,A -85,B 0,C 180,E1 -413.956,E2 -413.956} C_VEL
LIN {X 0,Y 608.45,Z 122.697,A -85,B 0,C 180,E1 -416.328,E2 -416.328} C_VEL
LIN {X 0,Y 608.446,Z 122.693,A -85,B 0,C 180,E1 -418.733,E2 -418.733} C_VEL
LIN {X 0,Y 608.434,Z 122.69,A -85,B 0,C 180,E1 -421.387,E2 -421.387} C_VEL
LIN {X 0,Y 608.432,Z 122.696,A -85,B 0,C 180,E1 -423.964,E2 -423.964} C_VEL
LIN {X 0,Y 608.43,Z 122.693,A -85,B 0,C 180,E1 -426.875,E2 -426.875} C_VEL
LIN {X 0,Y 608.435,Z 122.818,A -85,B 0,C 180,E1 -427.309,E2 -427.309} C_VEL
LIN {X 0,Y 608.573,Z 138.081,A -85,B 0,C 180,E1 -429.413,E2 -429.413} C_VEL
LIN {X 0,Y 608.533,Z 158.527,A -85,B 0,C 180,E1 -432.178,E2 -432.178} C_VEL
LIN {X 0,Y 608.493,Z 179.239,A -85,B 0,C 180,E1 -434.937,E2 -434.937} C_VEL
LIN {X 0,Y 608.441,Z 194.611,A -85,B 0,C 180,E1 -436.962,E2 -436.962} C_VEL
LIN {X 0,Y 608.569,Z 245.207,A -85,B 0,C 180,E1 -437.579,E2 -437.579} C_VEL
LIN {X 0,Y 608.547,Z 302.935,A -85,B 0,C 180,E1 -438.276,E2 -438.276} C_VEL
LIN {X 0,Y 608.512,Z 316.209,A -85,B 0,C 180,E1 -438.571,E2 -438.571} C_VEL
LIN {X 0,Y 608.514,Z 328.629,A -85,B 0,C 180,E1 -438.982,E2 -438.982} C_VEL
LIN {X 0,Y 608.499,Z 340.631,A -85,B 0,C 180,E1 -439.519,E2 -439.519} C_VEL
LIN {X 0,Y 608.484,Z 352.194,A -85,B 0,C 180,E1 -440.191,E2 -440.191} C_VEL
LIN {X 0,Y 608.485,Z 362.591,A -85,B 0,C 180,E1 -440.946,E2 -440.946} C_VEL
LIN {X 0,Y 608.475,Z 371.11,A -85,B 0,C 180,E1 -441.699,E2 -441.699} C_VEL
LIN {X 0,Y 608.471,Z 378.959,A -85,B 0,C 180,E1 -442.534,E2 -442.534} C_VEL
LIN {X 0,Y 608.461,Z 386.286,A -85,B 0,C 180,E1 -443.484,E2 -443.484} C_VEL
LIN {X 0,Y 608.451,Z 391.865,A -85,B 0,C 180,E1 -444.365,E2 -444.365} C_VEL
LIN {X 0,Y 608.432,Z 396.949,A -85,B 0,C 180,E1 -445.362,E2 -445.362} C_VEL
LIN {X 0,Y 608.449,Z 400.896,A -85,B 0,C 180,E1 -446.357,E2 -446.357} C_VEL
LIN {X 0,Y 608.425,Z 403.809,A -85,B 0,C 180,E1 -447.352,E2 -447.352} C_VEL
LIN {X 0,Y 608.445,Z 405.201,A -85,B 0,C 180,E1 -448.014,E2 -448.014} C_VEL
LIN {X 0,Y 608.438,Z 406.783,A -85,B 0,C 180,E1 -449.338,E2 -449.338} C_VEL
LIN {X 0,Y 608.434,Z 407,A -85,B 0,C 180,E1 -450,E2 -450} C_VEL
LIN {X 0,Y 608.448,Z 406.184,A -85,B 0,C 180,E1 -451.324,E2 -451.324} C_VEL
LIN {X 0,Y 608.445,Z 405.202,A -85,B 0,C 180,E1 -451.986,E2 -451.986} C_VEL
LIN {X 0,Y 608.425,Z 403.809,A -85,B 0,C 180,E1 -452.648,E2 -452.648} C_VEL
LIN {X 0,Y 608.449,Z 400.896,A -85,B 0,C 180,E1 -453.642,E2 -453.642} C_VEL
LIN {X 0,Y 608.432,Z 396.95,A -85,B 0,C 180,E1 -454.638,E2 -454.638} C_VEL
LIN {X 0,Y 608.438,Z 390.877,A -85,B 0,C 180,E1 -455.801,E2 -455.801} C_VEL
LIN {X 0,Y 608.462,Z 384.236,A -85,B 0,C 180,E1 -456.799,E2 -456.799} C_VEL
LIN {X 0,Y 608.456,Z 375.99,A -85,B 0,C 180,E1 -457.8,E2 -457.8} C_VEL
LIN {X 0,Y 608.472,Z 367.537,A -85,B 0,C 180,E1 -458.636,E2 -458.636} C_VEL
LIN {X 0,Y 608.479,Z 357.092,A -85,B 0,C 180,E1 -459.473,E2 -459.473} C_VEL
LIN {X 0,Y 608.489,Z 346.757,A -85,B 0,C 180,E1 -460.145,E2 -460.145} C_VEL
LIN {X 0,Y 608.519,Z 335.267,A -85,B 0,C 180,E1 -460.74,E2 -460.74} C_VEL
LIN {X 0,Y 608.528,Z 322.892,A -85,B 0,C 180,E1 -461.225,E2 -461.225} C_VEL
LIN {X 0,Y 608.544,Z 309.44,A -85,B 0,C 180,E1 -461.597,E2 -461.597} C_VEL
LIN {X 0,Y 608.553,Z 297.086,A -85,B 0,C 180,E1 -461.808,E2 -461.808} C_VEL
LIN {X 0,Y 608.496,Z 195.143,A -85,B 0,C 180,E1 -463.016,E2 -463.016} C_VEL
LIN {X 0,Y 608.444,Z 194.128,A -85,B 0,C 180,E1 -463.102,E2 -463.102} C_VEL
LIN {X 0,Y 608.497,Z 172.769,A -85,B 0,C 180,E1 -465.921,E2 -465.921} C_VEL
LIN {X 0,Y 608.499,Z 151.838,A -85,B 0,C 180,E1 -468.723,E2 -468.723} C_VEL
LIN {X 0,Y 608.575,Z 131.345,A -85,B 0,C 180,E1 -471.51,E2 -471.51} C_VEL
LIN {X 0,Y 608.425,Z 122.693,A -85,B 0,C 180,E1 -472.716,E2 -472.716} C_VEL
LIN {X 0,Y 608.438,Z 122.693,A -85,B 0,C 180,E1 -475.302,E2 -475.302} C_VEL
LIN {X 0,Y 608.436,Z 122.697,A -85,B 0,C 180,E1 -477.519,E2 -477.519} C_VEL
LIN {X 0,Y 608.43,Z 122.695,A -85,B 0,C 180,E1 -479.965,E2 -479.965} C_VEL
LIN {X 0,Y 608.418,Z 122.692,A -85,B 0,C 180,E1 -482.515,E2 -482.515} C_VEL
LIN {X 0,Y 608.419,Z 122.694,A -85,B 0,C 180,E1 -484.901,E2 -484.901} C_VEL
LIN {X 0,Y 608.439,Z 122.693,A -85,B 0,C 180,E1 -487.749,E2 -487.749} C_VEL
LIN {X 0,Y 608.404,Z 122.694,A -85,B 0,C 180,E1 -490.323,E2 -490.323} C_VEL
LIN {X 0,Y 608.444,Z 122.695,A -85,B 0,C 180,E1 -492.961,E2 -492.961} C_VEL
LIN {X 0,Y 608.407,Z 122.695,A -85,B 0,C 180,E1 -495.741,E2 -495.741} C_VEL
LIN {X 0,Y 608.405,Z 122.694,A -85,B 0,C 180,E1 -497.933,E2 -497.933} C_VEL
LIN {X 0,Y 608.434,Z 122.697,A -85,B 0,C 180,E1 -500.707,E2 -500.707} C_VEL
LIN {X 0,Y 608.432,Z 122.697,A -85,B 0,C 180,E1 -503.083,E2 -503.083} C_VEL
LIN {X 0,Y 608.392,Z 122.696,A -85,B 0,C 180,E1 -505.525,E2 -505.525} C_VEL
LIN {X 0,Y 608.411,Z 122.693,A -85,B 0,C 180,E1 -507.902,E2 -507.902} C_VEL
LIN {X 0,Y 608.431,Z 122.694,A -85,B 0,C 180,E1 -510.218,E2 -510.218} C_VEL
LIN {X 0,Y 608.397,Z 122.695,A -85,B 0,C 180,E1 -513.223,E2 -513.223} C_VEL
LIN {X 0,Y 608.409,Z 122.693,A -85,B 0,C 180,E1 -515.427,E2 -515.427} C_VEL
LIN {X 0,Y 608.452,Z 122.697,A -85,B 0,C 180,E1 -518.308,E2 -518.308} C_VEL
LIN {X 0,Y 608.414,Z 122.692,A -85,B 0,C 180,E1 -521.301,E2 -521.301} C_VEL
LIN {X 0,Y 608.439,Z 122.695,A -85,B 0,C 180,E1 -523.905,E2 -523.905} C_VEL
LIN {X 0,Y 608.436,Z 122.692,A -85,B 0,C 180,E1 -526.643,E2 -526.643} C_VEL
LIN {X 0,Y 608.42,Z 122.693,A -85,B 0,C 180,E1 -529.349,E2 -529.349} C_VEL
LIN {X 0,Y 608.476,Z 122.693,A -85,B 0,C 180,E1 -532.033,E2 -532.033} C_VEL
LIN {X 0,Y 608.426,Z 122.691,A -85,B 0,C 180,E1 -534.697,E2 -534.697} C_VEL
LIN {X 0,Y 608.45,Z 122.692,A -85,B 0,C 180,E1 -537.351,E2 -537.351} C_VEL
LIN {X 0,Y 608.478,Z 122.689,A -85,B 0,C 180,E1 -540,E2 -540} C_VEL
LIN {X 0,Y 608.44,Z 122.689,A -85,B 0,C 180,E1 -542.648,E2 -542.648} C_VEL
LIN {X 0,Y 608.454,Z 122.695,A -85,B 0,C 180,E1 -545.302,E2 -545.302} C_VEL
LIN {X 0,Y 608.472,Z 122.687,A -85,B 0,C 180,E1 -547.967,E2 -547.967} C_VEL
LIN {X 0,Y 608.459,Z 122.695,A -85,B 0,C 180,E1 -549.422,E2 -549.422} C_VEL
LIN {X 0,Y 607.777,Z 122.774,A -85,B 0,C 180,E1 -549.975,E2 -549.975} C_VEL
LIN {X 0,Y 604.925,Z 123.13,A -85,B 0,C 180,E1 -550.872,E2 -550.872} C_VEL
LIN {X 0,Y 602.519,Z 123.432,A -85,B 0,C 180,E1 -551.593,E2 -551.593} C_VEL
LIN {X 0,Y 601.478,Z 123.557,A -85,B 0,C 180,E1 -552.15,E2 -552.15} C_VEL
LIN {X 0,Y 601.388,Z 123.568,A -85,B 0,C 180,E1 -552.338,E2 -552.338} C_VEL
LIN {X 0,Y 601.4,Z 123.572,A -85,B 0,C 180,E1 -554.897,E2 -554.897} C_VEL
LIN {X 0,Y 601.41,Z 123.573,A -85,B 0,C 180,E1 -556.986,E2 -556.986} C_VEL
LIN {X 0,Y 601.396,Z 123.567,A -85,B 0,C 180,E1 -559.809,E2 -559.809} C_VEL
LIN {X 0,Y 601.404,Z 123.572,A -85,B 0,C 180,E1 -562.683,E2 -562.683} C_VEL
LIN {X 0,Y 601.429,Z 123.563,A -85,B 0,C 180,E1 -565.617,E2 -565.617} C_VEL
LIN {X 0,Y 601.394,Z 123.567,A -85,B 0,C 180,E1 -567.868,E2 -567.868} C_VEL
LIN {X 0,Y 601.405,Z 123.568,A -85,B 0,C 180,E1 -570.165,E2 -570.165} C_VEL
LIN {X 0,Y 601.42,Z 123.572,A -85,B 0,C 180,E1 -572.715,E2 -572.715} C_VEL
LIN {X 0,Y 601.395,Z 123.569,A -85,B 0,C 180,E1 -575.111,E2 -575.111} C_VEL
LIN {X 0,Y 601.435,Z 123.562,A -85,B 0,C 180,E1 -577.419,E2 -577.419} C_VEL
LIN {X 0,Y 601.4,Z 123.571,A -85,B 0,C 180,E1 -579.995,E2 -579.995} C_VEL
LIN {X 0,Y 601.415,Z 123.569,A -85,B 0,C 180,E1 -582.669,E2 -582.669} C_VEL
LIN {X 0,Y 601.425,Z 123.564,A -85,B 0,C 180,E1 -585.482,E2 -585.482} C_VEL
LIN {X 0,Y 601.423,Z 123.569,A -85,B 0,C 180,E1 -588.406,E2 -588.406} C_VEL
LIN {X 0,Y 601.458,Z 123.754,A -85,B 0,C 180,E1 -591.275,E2 -591.275} C_VEL
LIN {X 0,Y 601.465,Z 137.93,A -85,B 0,C 180,E1 -593.731,E2 -593.731} C_VEL
LIN {X 0,Y 601.416,Z 155.229,A -85,B 0,C 180,E1 -596.686,E2 -596.686} C_VEL
LIN {X 0,Y 601.439,Z 156.38,A -85,B 0,C 180,E1 -596.881,E2 -596.881} C_VEL
LIN {X 0,Y 601.677,Z 163.617,A -85,B 0,C 180,E1 -596.981,E2 -596.981} C_VEL
LIN {X 0,Y 601.589,Z 263.027,A -85,B 0,C 180,E1 -598.186,E2 -598.186} C_VEL
LIN {X 0,Y 601.586,Z 276.17,A -85,B 0,C 180,E1 -598.482,E2 -598.482} C_VEL
LIN {X 0,Y 601.546,Z 288.606,A -85,B 0,C 180,E1 -598.897,E2 -598.897} C_VEL
LIN {X 0,Y 601.482,Z 300.829,A -85,B 0,C 180,E1 -599.451,E2 -599.451} C_VEL
LIN {X 0,Y 601.444,Z 312.299,A -85,B 0,C 180,E1 -600.127,E2 -600.127} C_VEL
LIN {X 0,Y 601.457,Z 323.344,A -85,B 0,C 180,E1 -600.944,E2 -600.944} C_VEL
LIN {X 0,Y 601.416,Z 332.192,A -85,B 0,C 180,E1 -601.753,E2 -601.753} C_VEL
LIN {X 0,Y 601.399,Z 340.173,A -85,B 0,C 180,E1 -602.64,E2 -602.64} C_VEL
LIN {X 0,Y 601.383,Z 347.502,A -85,B 0,C 180,E1 -603.635,E2 -603.635} C_VEL
LIN {X 0,Y 601.373,Z 354.057,A -85,B 0,C 180,E1 -604.75,E2 -604.75} C_VEL
LIN {X 0,Y 601.354,Z 359.054,A -85,B 0,C 180,E1 -605.855,E2 -605.855} C_VEL
LIN {X 0,Y 601.353,Z 362.717,A -85,B 0,C 180,E1 -606.951,E2 -606.951} C_VEL
LIN {X 0,Y 601.336,Z 365.206,A -85,B 0,C 180,E1 -608.038,E2 -608.038} C_VEL
LIN {X 0,Y 601.34,Z 366.678,A -85,B 0,C 180,E1 -609.223,E2 -609.223} C_VEL
LIN {X 0,Y 601.314,Z 366.973,A -85,B 0,C 180,E1 -610.187,E2 -610.187} C_VEL
LIN {X 0,Y 601.341,Z 366.398,A -85,B 0,C 180,E1 -611.201,E2 -611.201} C_VEL
LIN {X 0,Y 601.312,Z 364.712,A -85,B 0,C 180,E1 -612.309,E2 -612.309} C_VEL
LIN {X 0,Y 601.333,Z 361.92,A -85,B 0,C 180,E1 -613.407,E2 -613.407} C_VEL
LIN {X 0,Y 601.338,Z 358.35,A -85,B 0,C 180,E1 -614.407,E2 -614.407} C_VEL
LIN {X 0,Y 601.338,Z 353.48,A -85,B 0,C 180,E1 -615.447,E2 -615.447} C_VEL
LIN {X 0,Y 601.37,Z 347.315,A -85,B 0,C 180,E1 -616.483,E2 -616.483} C_VEL
LIN {X 0,Y 601.396,Z 339.657,A -85,B 0,C 180,E1 -617.514,E2 -617.514} C_VEL
LIN {X 0,Y 601.431,Z 331.861,A -85,B 0,C 180,E1 -618.371,E2 -618.371} C_VEL
LIN {X 0,Y 601.437,Z 322.37,A -85,B 0,C 180,E1 -619.224,E2 -619.224} C_VEL
LIN {X 0,Y 601.471,Z 311.88,A -85,B 0,C 180,E1 -619.991,E2 -619.991} C_VEL
LIN {X 0,Y 601.519,Z 300.219,A -85,B 0,C 180,E1 -620.671,E2 -620.671} C_VEL
LIN {X 0,Y 601.535,Z 287.86,A -85,B 0,C 180,E1 -621.222,E2 -621.222} C_VEL
LIN {X 0,Y 601.536,Z 274.908,A -85,B 0,C 180,E1 -621.645,E2 -621.645} C_VEL
LIN {X 0,Y 601.593,Z 262.098,A -85,B 0,C 180,E1 -621.92,E2 -621.92} C_VEL
LIN {X 0,Y 601.561,Z 157.7,A -85,B 0,C 180,E1 -623.183,E2 -623.183} C_VEL
LIN {X 0,Y 601.379,Z 156.408,A -85,B 0,C 180,E1 -623.205,E2 -623.205} C_VEL
LIN {X 0,Y 601.422,Z 142.102,A -85,B 0,C 180,E1 -625.644,E2 -625.644} C_VEL
LIN {X 0,Y 601.452,Z 124.641,A -85,B 0,C 180,E1 -628.661,E2 -628.661} C_VEL
LIN {X 0,Y 601.368,Z 123.573,A -85,B 0,C 180,E1 -628.87,E2 -628.87} C_VEL
LIN {X 0,Y 601.363,Z 123.573,A -85,B 0,C 180,E1 -630.67,E2 -630.67} C_VEL
LIN {X 0,Y 601.393,Z 123.569,A -85,B 0,C 180,E1 -632.679,E2 -632.679} C_VEL
LIN {X 0,Y 601.384,Z 123.57,A -85,B 0,C 180,E1 -635.365,E2 -635.365} C_VEL
LIN {X 0,Y 601.423,Z 123.571,A -85,B 0,C 180,E1 -638.061,E2 -638.061} C_VEL
LIN {X 0,Y 601.37,Z 123.57,A -85,B 0,C 180,E1 -640.987,E2 -640.987} C_VEL
LIN {X 0,Y 601.381,Z 123.575,A -85,B 0,C 180,E1 -643.517,E2 -643.517} C_VEL
LIN {X 0,Y 601.383,Z 123.57,A -85,B 0,C 180,E1 -646.289,E2 -646.289} C_VEL
LIN {X 0,Y 601.362,Z 123.573,A -85,B 0,C 180,E1 -649.101,E2 -649.101} C_VEL
LIN {X 0,Y 601.382,Z 123.573,A -85,B 0,C 180,E1 -651.241,E2 -651.241} C_VEL
LIN {X 0,Y 601.374,Z 123.57,A -85,B 0,C 180,E1 -654.28,E2 -654.28} C_VEL
LIN {X 0,Y 601.405,Z 123.571,A -85,B 0,C 180,E1 -657.114,E2 -657.114} C_VEL
LIN {X 0,Y 601.37,Z 123.58,A -85,B 0,C 180,E1 -659.396,E2 -659.396} C_VEL
LIN {X 0,Y 601.371,Z 123.573,A -85,B 0,C 180,E1 -661.729,E2 -661.729} C_VEL
LIN {X 0,Y 601.374,Z 123.569,A -85,B 0,C 180,E1 -664.122,E2 -664.122} C_VEL
LIN {X 0,Y 601.4,Z 123.572,A -85,B 0,C 180,E1 -667.378,E2 -667.378} C_VEL
LIN {X 0,Y 601.371,Z 123.57,A -85,B 0,C 180,E1 -669.999,E2 -669.999} C_VEL
LIN {X 0,Y 601.364,Z 123.575,A -85,B 0,C 180,E1 -672.675,E2 -672.675} C_VEL
LIN {X 0,Y 601.398,Z 123.569,A -85,B 0,C 180,E1 -675.48,E2 -675.48} C_VEL
LIN {X 0,Y 601.383,Z 123.571,A -85,B 0,C 180,E1 -678.412,E2 -678.412} C_VEL
LIN {X 0,Y 601.393,Z 123.577,A -85,B 0,C 180,E1 -680.873,E2 -680.873} C_VEL
LIN {X 0,Y 601.377,Z 123.57,A -85,B 0,C 180,E1 -683.416,E2 -683.416} C_VEL
LIN {X 0,Y 601.382,Z 123.57,A -85,B 0,C 180,E1 -686.072,E2 -686.072} C_VEL
LIN {X 0,Y 601.391,Z 123.577,A -85,B 0,C 180,E1 -688.551,E2 -688.551} C_VEL
LIN {X 0,Y 601.381,Z 123.569,A -85,B 0,C 180,E1 -691.371,E2 -691.371} C_VEL
LIN {X 0,Y 601.394,Z 123.572,A -85,B 0,C 180,E1 -694.138,E2 -694.138} C_VEL
LIN {X 0,Y 601.371,Z 123.577,A -85,B 0,C 180,E1 -696.588,E2 -696.588} C_VEL
LIN {X 0,Y 601.386,Z 123.568,A -85,B 0,C 180,E1 -699.477,E2 -699.477} C_VEL
LIN {X 0,Y 601.371,Z 123.58,A -85,B 0,C 180,E1 -702.311,E2 -702.311} C_VEL
LIN {X 0,Y 601.373,Z 123.57,A -85,B 0,C 180,E1 -705.102,E2 -705.102} C_VEL
LIN {X 0,Y 601.395,Z 123.572,A -85,B 0,C 180,E1 -707.857,E2 -707.857} C_VEL
LIN {X 0,Y 601.385,Z 123.57,A -85,B 0,C 180,E1 -710.584,E2 -710.584} C_VEL
LIN {X 0,Y 601.375,Z 123.571,A -85,B 0,C 180,E1 -712.614,E2 -712.614} C_VEL
LIN {X 0,Y 601.389,Z 123.569,A -85,B 0,C 180,E1 -714.636,E2 -714.636} C_VEL
LIN {X 0,Y 601.402,Z 123.568,A -85,B 0,C 180,E1 -717.321,E2 -717.321} C_VEL
LIN {X 0,Y 601.446,Z 123.568,A -85,B 0,C 180,E1 -720,E2 -720} C_VEL
LIN {X 0,Y 601.395,Z 123.567,A -85,B 0,C 180,E1 -722.68,E2 -722.68} C_VEL
LIN {X 0,Y 601.4,Z 123.571,A -85,B 0,C 180,E1 -725.365,E2 -725.365} C_VEL
LIN {X 0,Y 601.429,Z 123.566,A -85,B 0,C 180,E1 -728.061,E2 -728.061} C_VEL
LIN {X 0,Y 601.397,Z 123.568,A -85,B 0,C 180,E1 -730.995,E2 -730.995} C_VEL
LIN {X 0,Y 601.394,Z 123.577,A -85,B 0,C 180,E1 -733.517,E2 -733.517} C_VEL
LIN {X 0,Y 601.391,Z 123.567,A -85,B 0,C 180,E1 -736.289,E2 -736.289} C_VEL
LIN {X 0,Y 601.407,Z 123.571,A -85,B 0,C 180,E1 -739.1,E2 -739.1} C_VEL
LIN {X 0,Y 601.381,Z 123.57,A -85,B 0,C 180,E1 -741.961,E2 -741.961} C_VEL
LIN {X 0,Y 601.384,Z 123.573,A -85,B 0,C 180,E1 -744.88,E2 -744.88} C_VEL
LIN {X 0,Y 601.412,Z 123.571,A -85,B 0,C 180,E1 -747.361,E2 -747.361} C_VEL
LIN {X 0,Y 601.377,Z 123.569,A -85,B 0,C 180,E1 -750.167,E2 -750.167} C_VEL
LIN {X 0,Y 601.398,Z 123.571,A -85,B 0,C 180,E1 -752.711,E2 -752.711} C_VEL
LIN {X 0,Y 601.385,Z 123.576,A -85,B 0,C 180,E1 -755.11,E2 -755.11} C_VEL
LIN {X 0,Y 601.434,Z 123.564,A -85,B 0,C 180,E1 -757.419,E2 -757.419} C_VEL
LIN {X 0,Y 601.379,Z 123.569,A -85,B 0,C 180,E1 -759.998,E2 -759.998} C_VEL
LIN {X 0,Y 601.381,Z 123.577,A -85,B 0,C 180,E1 -762.673,E2 -762.673} C_VEL
LIN {X 0,Y 601.404,Z 123.566,A -85,B 0,C 180,E1 -765.479,E2 -765.479} C_VEL
LIN {X 0,Y 601.417,Z 123.571,A -85,B 0,C 180,E1 -768.408,E2 -768.408} C_VEL
LIN {X 0,Y 601.402,Z 123.571,A -85,B 0,C 180,E1 -770.872,E2 -770.872} C_VEL
LIN {X 0,Y 601.391,Z 123.567,A -85,B 0,C 180,E1 -773.416,E2 -773.416} C_VEL
LIN {X 0,Y 601.415,Z 123.569,A -85,B 0,C 180,E1 -776.067,E2 -776.067} C_VEL
LIN {X 0,Y 601.395,Z 123.568,A -85,B 0,C 180,E1 -779.056,E2 -779.056} C_VEL
LIN {X 0,Y 601.395,Z 123.567,A -85,B 0,C 180,E1 -781.371,E2 -781.371} C_VEL
LIN {X 0,Y 601.411,Z 123.574,A -85,B 0,C 180,E1 -784.134,E2 -784.134} C_VEL
LIN {X 0,Y 601.404,Z 123.57,A -85,B 0,C 180,E1 -787.044,E2 -787.044} C_VEL
LIN {X 0,Y 601.379,Z 123.577,A -85,B 0,C 180,E1 -787.134,E2 -787.134} C_VEL
LIN {X 0,Y 601.667,Z 130.049,A -85,B 0,C 180,E1 -788.05,E2 -788.05} C_VEL
LIN {X 0,Y 601.598,Z 150.761,A -85,B 0,C 180,E1 -790.907,E2 -790.907} C_VEL
LIN {X 0,Y 601.519,Z 172.767,A -85,B 0,C 180,E1 -793.889,E2 -793.889} C_VEL
LIN {X 0,Y 601.449,Z 194.449,A -85,B 0,C 180,E1 -796.786,E2 -796.786} C_VEL
LIN {X 0,Y 601.612,Z 196.017,A -85,B 0,C 180,E1 -796.843,E2 -796.843} C_VEL
LIN {X 0,Y 601.614,Z 302.935,A -85,B 0,C 180,E1 -798.139,E2 -798.139} C_VEL
LIN {X 0,Y 601.56,Z 316.21,A -85,B 0,C 180,E1 -798.437,E2 -798.437} C_VEL
LIN {X 0,Y 601.546,Z 327.901,A -85,B 0,C 180,E1 -798.825,E2 -798.825} C_VEL
LIN {X 0,Y 601.523,Z 340.629,A -85,B 0,C 180,E1 -799.396,E2 -799.396} C_VEL
LIN {X 0,Y 601.483,Z 352.196,A -85,B 0,C 180,E1 -800.076,E2 -800.076} C_VEL
LIN {X 0,Y 601.444,Z 362.593,A -85,B 0,C 180,E1 -800.839,E2 -800.839} C_VEL
LIN {X 0,Y 601.429,Z 371.11,A -85,B 0,C 180,E1 -801.601,E2 -801.601} C_VEL
LIN {X 0,Y 601.418,Z 378.959,A -85,B 0,C 180,E1 -802.446,E2 -802.446} C_VEL
LIN {X 0,Y 601.37,Z 386.224,A -85,B 0,C 180,E1 -803.398,E2 -803.398} C_VEL
LIN {X 0,Y 601.372,Z 391.865,A -85,B 0,C 180,E1 -804.299,E2 -804.299} C_VEL
LIN {X 0,Y 601.336,Z 396.949,A -85,B 0,C 180,E1 -805.307,E2 -805.307} C_VEL
LIN {X 0,Y 601.368,Z 400.895,A -85,B 0,C 180,E1 -806.315,E2 -806.315} C_VEL
LIN {X 0,Y 601.325,Z 403.809,A -85,B 0,C 180,E1 -807.32,E2 -807.32} C_VEL
LIN {X 0,Y 601.343,Z 405.201,A -85,B 0,C 180,E1 -807.991,E2 -807.991} C_VEL
LIN {X 0,Y 601.339,Z 406.784,A -85,B 0,C 180,E1 -809.33,E2 -809.33} C_VEL
LIN {X 0,Y 601.335,Z 407,A -85,B 0,C 180,E1 -810,E2 -810} C_VEL
LIN {X 0,Y 601.347,Z 406.185,A -85,B 0,C 180,E1 -811.339,E2 -811.339} C_VEL
LIN {X 0,Y 601.343,Z 405.202,A -85,B 0,C 180,E1 -812.009,E2 -812.009} C_VEL
LIN {X 0,Y 601.325,Z 403.81,A -85,B 0,C 180,E1 -812.679,E2 -812.679} C_VEL
LIN {X 0,Y 601.368,Z 400.896,A -85,B 0,C 180,E1 -813.685,E2 -813.685} C_VEL
LIN {X 0,Y 601.336,Z 396.95,A -85,B 0,C 180,E1 -814.693,E2 -814.693} C_VEL
LIN {X 0,Y 601.373,Z 390.878,A -85,B 0,C 180,E1 -815.869,E2 -815.869} C_VEL
LIN {X 0,Y 601.382,Z 384.236,A -85,B 0,C 180,E1 -816.88,E2 -816.88} C_VEL
LIN {X 0,Y 601.4,Z 375.99,A -85,B 0,C 180,E1 -817.892,E2 -817.892} C_VEL
LIN {X 0,Y 601.436,Z 367.537,A -85,B 0,C 180,E1 -818.738,E2 -818.738} C_VEL
LIN {X 0,Y 601.449,Z 357.094,A -85,B 0,C 180,E1 -819.585,E2 -819.585} C_VEL
LIN {X 0,Y 601.467,Z 346.759,A -85,B 0,C 180,E1 -820.264,E2 -820.264} C_VEL
LIN {X 0,Y 601.538,Z 334.599,A -85,B 0,C 180,E1 -820.896,E2 -820.896} C_VEL
LIN {X 0,Y 601.555,Z 322.219,A -85,B 0,C 180,E1 -821.379,E2 -821.379} C_VEL
LIN {X 0,Y 601.583,Z 309.438,A -85,B 0,C 180,E1 -821.733,E2 -821.733} C_VEL
LIN {X 0,Y 601.62,Z 297.086,A -85,B 0,C 180,E1 -821.946,E2 -821.946} C_VEL
LIN {X 0,Y 601.471,Z 195.143,A -85,B 0,C 180,E1 -823.171,E2 -823.171} C_VEL
LIN {X 0,Y 601.455,Z 194.128,A -85,B 0,C 180,E1 -823.257,E2 -823.257} C_VEL
LIN {X 0,Y 601.519,Z 172.769,A -85,B 0,C 180,E1 -826.11,E2 -826.11} C_VEL
LIN {X 0,Y 601.598,Z 150.762,A -85,B 0,C 180,E1 -829.093,E2 -829.093} C_VEL
LIN {X 0,Y 601.651,Z 131.345,A -85,B 0,C 180,E1 -831.77,E2 -831.77} C_VEL
LIN {X 0,Y 601.591,Z 124.873,A -85,B 0,C 180,E1 -832.676,E2 -832.676} C_VEL
LIN {X 0,Y 601.393,Z 123.571,A -85,B 0,C 180,E1 -832.888,E2 -832.888} C_VEL
LIN {X 0,Y 601.422,Z 123.572,A -85,B 0,C 180,E1 -835.618,E2 -835.618} C_VEL
LIN {X 0,Y 601.367,Z 123.578,A -85,B 0,C 180,E1 -837.87,E2 -837.87} C_VEL
LIN {X 0,Y 601.4,Z 123.569,A -85,B 0,C 180,E1 -840.166,E2 -840.166} C_VEL
LIN {X 0,Y 601.392,Z 123.568,A -85,B 0,C 180,E1 -842.71,E2 -842.71} C_VEL
LIN {X 0,Y 601.374,Z 123.574,A -85,B 0,C 180,E1 -845.109,E2 -845.109} C_VEL
LIN {X 0,Y 601.432,Z 123.572,A -85,B 0,C 180,E1 -847.419,E2 -847.419} C_VEL
LIN {X 0,Y 601.377,Z 123.57,A -85,B 0,C 180,E1 -849.998,E2 -849.998} C_VEL
LIN {X 0,Y 601.369,Z 123.573,A -85,B 0,C 180,E1 -852.674,E2 -852.674} C_VEL
LIN {X 0,Y 601.402,Z 123.57,A -85,B 0,C 180,E1 -855.479,E2 -855.479} C_VEL
LIN {X 0,Y 601.385,Z 123.57,A -85,B 0,C 180,E1 -858.411,E2 -858.411} C_VEL
LIN {X 0,Y 601.395,Z 123.577,A -85,B 0,C 180,E1 -860.872,E2 -860.872} C_VEL
LIN {X 0,Y 601.372,Z 123.572,A -85,B 0,C 180,E1 -863.415,E2 -863.415} C_VEL
LIN {X 0,Y 601.363,Z 123.572,A -85,B 0,C 180,E1 -866.075,E2 -866.075} C_VEL
LIN {X 0,Y 601.39,Z 123.576,A -85,B 0,C 180,E1 -868.551,E2 -868.551} C_VEL
LIN {X 0,Y 601.38,Z 123.569,A -85,B 0,C 180,E1 -871.37,E2 -871.37} C_VEL
LIN {X 0,Y 601.393,Z 123.571,A -85,B 0,C 180,E1 -874.137,E2 -874.137} C_VEL
LIN {X 0,Y 601.372,Z 123.577,A -85,B 0,C 180,E1 -876.587,E2 -876.587} C_VEL
LIN {X 0,Y 601.389,Z 123.568,A -85,B 0,C 180,E1 -879.476,E2 -879.476} C_VEL
LIN {X 0,Y 601.374,Z 123.578,A -85,B 0,C 180,E1 -882.311,E2 -882.311} C_VEL
LIN {X 0,Y 601.377,Z 123.569,A -85,B 0,C 180,E1 -885.101,E2 -885.101} C_VEL
LIN {X 0,Y 601.402,Z 123.573,A -85,B 0,C 180,E1 -887.857,E2 -887.857} C_VEL
LIN {X 0,Y 601.39,Z 123.569,A -85,B 0,C 180,E1 -890.583,E2 -890.583} C_VEL
LIN {X 0,Y 601.379,Z 123.57,A -85,B 0,C 180,E1 -892.614,E2 -892.614} C_VEL
LIN {X 0,Y 601.392,Z 123.57,A -85,B 0,C 180,E1 -895.307,E2 -895.307} C_VEL
LIN {X 0,Y 601.436,Z 123.567,A -85,B 0,C 180,E1 -897.991,E2 -897.991} C_VEL
LIN {X 0,Y 601.396,Z 123.566,A -85,B 0,C 180,E1 -900.669,E2 -900.669} C_VEL
LIN {X 0,Y 601.416,Z 123.571,A -85,B 0,C 180,E1 -903.349,E2 -903.349} C_VEL
LIN {X 0,Y 601.413,Z 123.566,A -85,B 0,C 180,E1 -906.037,E2 -906.037} C_VEL
LIN {X 0,Y 601.393,Z 123.569,A -85,B 0,C 180,E1 -908.738,E2 -908.738} C_VEL
LIN {X 0,Y 601.435,Z 123.569,A -85,B 0,C 180,E1 -911.458,E2 -911.458} C_VEL
LIN {X 0,Y 601.388,Z 123.568,A -85,B 0,C 180,E1 -912.338,E2 -912.338} C_VEL
LIN {X 0,Y 600.709,Z 123.658,A -85,B 0,C 180,E1 -912.897,E2 -912.897} C_VEL
LIN {X 0,Y 597.859,Z 124.017,A -85,B 0,C 180,E1 -913.805,E2 -913.805} C_VEL
LIN {X 0,Y 595.459,Z 124.317,A -85,B 0,C 180,E1 -914.536,E2 -914.536} C_VEL
LIN {X 0,Y 594.43,Z 124.444,A -85,B 0,C 180,E1 -915.099,E2 -915.099} C_VEL
LIN {X 0,Y 594.347,Z 124.45,A -85,B 0,C 180,E1 -915.29,E2 -915.29} C_VEL
LIN {X 0,Y 594.34,Z 124.446,A -85,B 0,C 180,E1 -917.905,E2 -917.905} C_VEL
LIN {X 0,Y 594.393,Z 124.446,A -85,B 0,C 180,E1 -920.776,E2 -920.776} C_VEL
LIN {X 0,Y 594.357,Z 124.444,A -85,B 0,C 180,E1 -923.705,E2 -923.705} C_VEL
LIN {X 0,Y 594.378,Z 124.442,A -85,B 0,C 180,E1 -926.02,E2 -926.02} C_VEL
LIN {X 0,Y 594.38,Z 124.446,A -85,B 0,C 180,E1 -928.998,E2 -928.998} C_VEL
LIN {X 0,Y 594.374,Z 124.442,A -85,B 0,C 180,E1 -931.642,E2 -931.642} C_VEL
LIN {X 0,Y 594.379,Z 124.451,A -85,B 0,C 180,E1 -934.58,E2 -934.58} C_VEL
LIN {X 0,Y 594.389,Z 124.441,A -85,B 0,C 180,E1 -937.608,E2 -937.608} C_VEL
LIN {X 0,Y 594.368,Z 124.449,A -85,B 0,C 180,E1 -940.566,E2 -940.566} C_VEL
LIN {X 0,Y 594.367,Z 124.443,A -85,B 0,C 180,E1 -943.299,E2 -943.299} C_VEL
LIN {X 0,Y 594.368,Z 124.453,A -85,B 0,C 180,E1 -946.16,E2 -946.16} C_VEL
LIN {X 0,Y 594.377,Z 124.442,A -85,B 0,C 180,E1 -949.177,E2 -949.177} C_VEL
LIN {X 0,Y 594.43,Z 124.627,A -85,B 0,C 180,E1 -951.198,E2 -951.198} C_VEL
LIN {X 0,Y 594.428,Z 139.243,A -85,B 0,C 180,E1 -953.761,E2 -953.761} C_VEL
LIN {X 0,Y 594.385,Z 155.935,A -85,B 0,C 180,E1 -956.646,E2 -956.646} C_VEL
LIN {X 0,Y 594.367,Z 156.474,A -85,B 0,C 180,E1 -956.73,E2 -956.73} C_VEL
LIN {X 0,Y 594.757,Z 161.152,A -85,B 0,C 180,E1 -956.796,E2 -956.796} C_VEL
LIN {X 0,Y 594.657,Z 263.414,A -85,B 0,C 180,E1 -958.053,E2 -958.053} C_VEL
LIN {X 0,Y 594.62,Z 276.627,A -85,B 0,C 180,E1 -958.357,E2 -958.357} C_VEL
LIN {X 0,Y 594.562,Z 289.766,A -85,B 0,C 180,E1 -958.809,E2 -958.809} C_VEL
LIN {X 0,Y 594.485,Z 301.25,A -85,B 0,C 180,E1 -959.348,E2 -959.348} C_VEL
LIN {X 0,Y 594.438,Z 312.935,A -85,B 0,C 180,E1 -960.051,E2 -960.051} C_VEL
LIN {X 0,Y 594.409,Z 323.024,A -85,B 0,C 180,E1 -960.809,E2 -960.809} C_VEL
LIN {X 0,Y 594.381,Z 331.476,A -85,B 0,C 180,E1 -961.581,E2 -961.581} C_VEL
LIN {X 0,Y 594.328,Z 340.06,A -85,B 0,C 180,E1 -962.537,E2 -962.537} C_VEL
LIN {X 0,Y 594.291,Z 348.266,A -85,B 0,C 180,E1 -963.675,E2 -963.675} C_VEL
LIN {X 0,Y 594.294,Z 354.637,A -85,B 0,C 180,E1 -964.803,E2 -964.803} C_VEL
LIN {X 0,Y 594.278,Z 359.564,A -85,B 0,C 180,E1 -965.945,E2 -965.945} C_VEL
LIN {X 0,Y 594.246,Z 363.015,A -85,B 0,C 180,E1 -967.028,E2 -967.028} C_VEL
LIN {X 0,Y 594.25,Z 364.73,A -85,B 0,C 180,E1 -967.762,E2 -967.762} C_VEL
LIN {X 0,Y 594.226,Z 365.954,A -85,B 0,C 180,E1 -968.491,E2 -968.491} C_VEL
LIN {X 0,Y 594.253,Z 366.682,A -85,B 0,C 180,E1 -969.219,E2 -969.219} C_VEL
LIN {X 0,Y 594.218,Z 366.982,A -85,B 0,C 180,E1 -969.941,E2 -969.941} C_VEL
LIN {X 0,Y 594.24,Z 366.511,A -85,B 0,C 180,E1 -971.11,E2 -971.11} C_VEL
LIN {X 0,Y 594.207,Z 365.181,A -85,B 0,C 180,E1 -972.09,E2 -972.09} C_VEL
LIN {X 0,Y 594.246,Z 362.293,A -85,B 0,C 180,E1 -973.327,E2 -973.327} C_VEL
LIN {X 0,Y 594.263,Z 357.894,A -85,B 0,C 180,E1 -974.568,E2 -974.568} C_VEL
LIN {X 0,Y 594.268,Z 352.903,A -85,B 0,C 180,E1 -975.62,E2 -975.62} C_VEL
LIN {X 0,Y 594.3,Z 346.609,A -85,B 0,C 180,E1 -976.668,E2 -976.668} C_VEL
LIN {X 0,Y 594.348,Z 338.779,A -85,B 0,C 180,E1 -977.711,E2 -977.711} C_VEL
LIN {X 0,Y 594.367,Z 330.68,A -85,B 0,C 180,E1 -978.586,E2 -978.586} C_VEL
LIN {X 0,Y 594.426,Z 319.981,A -85,B 0,C 180,E1 -979.527,E2 -979.527} C_VEL
LIN {X 0,Y 594.478,Z 308.893,A -85,B 0,C 180,E1 -980.301,E2 -980.301} C_VEL
LIN {X 0,Y 594.534,Z 298.077,A -85,B 0,C 180,E1 -980.903,E2 -980.903} C_VEL
LIN {X 0,Y 594.596,Z 286.187,A -85,B 0,C 180,E1 -981.418,E2 -981.418} C_VEL
LIN {X 0,Y 594.623,Z 273.331,A -85,B 0,C 180,E1 -981.825,E2 -981.825} C_VEL
LIN {X 0,Y 594.638,Z 260.689,A -85,B 0,C 180,E1 -982.082,E2 -982.082} C_VEL
LIN {X 0,Y 594.619,Z 158.109,A -85,B 0,C 180,E1 -983.334,E2 -983.334} C_VEL
LIN {X 0,Y 594.356,Z 156.313,A -85,B 0,C 180,E1 -983.38,E2 -983.38} C_VEL
LIN {X 0,Y 594.386,Z 141.535,A -85,B 0,C 180,E1 -985.932,E2 -985.932} C_VEL
LIN {X 0,Y 594.435,Z 125.062,A -85,B 0,C 180,E1 -988.815,E2 -988.815} C_VEL
LIN {X 0,Y 594.32,Z 124.452,A -85,B 0,C 180,E1 -988.984,E2 -988.984} C_VEL
LIN {X 0,Y 594.318,Z 124.451,A -85,B 0,C 180,E1 -990.678,E2 -990.678} C_VEL
LIN {X 0,Y 594.36,Z 124.445,A -85,B 0,C 180,E1 -992.711,E2 -992.711} C_VEL
LIN {X 0,Y 594.354,Z 124.446,A -85,B 0,C 180,E1 -995.428,E2 -995.428} C_VEL
LIN {X 0,Y 594.365,Z 124.448,A -85,B 0,C 180,E1 -998.158,E2 -998.158} C_VEL
LIN {X 0,Y 594.326,Z 124.448,A -85,B 0,C 180,E1 -1001.044,E2 -1001.044} C_VEL
LIN {X 0,Y 594.349,Z 124.454,A -85,B 0,C 180,E1 -1003.68,E2 -1003.68} C_VEL
LIN {X 0,Y 594.312,Z 124.449,A -85,B 0,C 180,E1 -1006.694,E2 -1006.694} C_VEL
LIN {X 0,Y 594.328,Z 124.453,A -85,B 0,C 180,E1 -1009.336,E2 -1009.336} C_VEL
LIN {X 0,Y 594.337,Z 124.456,A -85,B 0,C 180,E1 -1011.505,E2 -1011.505} C_VEL
LIN {X 0,Y 594.335,Z 124.446,A -85,B 0,C 180,E1 -1014.449,E2 -1014.449} C_VEL
LIN {X 0,Y 594.344,Z 124.446,A -85,B 0,C 180,E1 -1016.702,E2 -1016.702} C_VEL
LIN {X 0,Y 594.327,Z 124.451,A -85,B 0,C 180,E1 -1019.779,E2 -1019.779} C_VEL
LIN {X 0,Y 594.327,Z 124.447,A -85,B 0,C 180,E1 -1022.15,E2 -1022.15} C_VEL
LIN {X 0,Y 594.342,Z 124.447,A -85,B 0,C 180,E1 -1024.583,E2 -1024.583} C_VEL
LIN {X 0,Y 594.351,Z 124.447,A -85,B 0,C 180,E1 -1027.604,E2 -1027.604} C_VEL
LIN {X 0,Y 594.336,Z 124.449,A -85,B 0,C 180,E1 -1030.57,E2 -1030.57} C_VEL
LIN {X 0,Y 594.337,Z 124.451,A -85,B 0,C 180,E1 -1033.303,E2 -1033.303} C_VEL
LIN {X 0,Y 594.34,Z 124.446,A -85,B 0,C 180,E1 -1036.164,E2 -1036.164} C_VEL
LIN {X 0,Y 594.355,Z 124.449,A -85,B 0,C 180,E1 -1039.181,E2 -1039.181} C_VEL
LIN {X 0,Y 594.342,Z 124.446,A -85,B 0,C 180,E1 -1042.057,E2 -1042.057} C_VEL
LIN {X 0,Y 594.309,Z 124.459,A -85,B 0,C 180,E1 -1044.683,E2 -1044.683} C_VEL
LIN {X 0,Y 594.34,Z 124.449,A -85,B 0,C 180,E1 -1047.095,E2 -1047.095} C_VEL
LIN {X 0,Y 594.346,Z 124.445,A -85,B 0,C 180,E1 -1049.68,E2 -1049.68} C_VEL
LIN {X 0,Y 594.338,Z 124.456,A -85,B 0,C 180,E1 -1052.538,E2 -1052.538} C_VEL
LIN {X 0,Y 594.332,Z 124.451,A -85,B 0,C 180,E1 -1054.805,E2 -1054.805} C_VEL
LIN {X 0,Y 594.306,Z 124.45,A -85,B 0,C 180,E1 -1057.28,E2 -1057.28} C_VEL
LIN {X 0,Y 594.345,Z 124.449,A -85,B 0,C 180,E1 -1059.946,E2 -1059.946} C_VEL
LIN {X 0,Y 594.322,Z 124.45,A -85,B 0,C 180,E1 -1062.805,E2 -1062.805} C_VEL
LIN {X 0,Y 594.353,Z 124.446,A -85,B 0,C 180,E1 -1065.622,E2 -1065.622} C_VEL
LIN {X 0,Y 594.371,Z 124.447,A -85,B 0,C 180,E1 -1068.404,E2 -1068.404} C_VEL
LIN {X 0,Y 594.327,Z 124.447,A -85,B 0,C 180,E1 -1071.157,E2 -1071.157} C_VEL
LIN {X 0,Y 594.361,Z 124.452,A -85,B 0,C 180,E1 -1073.891,E2 -1073.891} C_VEL
LIN {X 0,Y 594.315,Z 124.45,A -85,B 0,C 180,E1 -1076.611,E2 -1076.611} C_VEL
LIN {X 0,Y 594.337,Z 124.446,A -85,B 0,C 180,E1 -1078.645,E2 -1078.645} C_VEL
LIN {X 0,Y 594.32,Z 124.448,A -85,B 0,C 180,E1 -1080.678,E2 -1080.678} C_VEL
LIN {X 0,Y 594.364,Z 124.443,A -85,B 0,C 180,E1 -1082.711,E2 -1082.711} C_VEL
LIN {X 0,Y 594.368,Z 124.448,A -85,B 0,C 180,E1 -1085.428,E2 -1085.428} C_VEL
LIN {X 0,Y 594.373,Z 124.444,A -85,B 0,C 180,E1 -1088.158,E2 -1088.158} C_VEL
LIN {X 0,Y 594.371,Z 124.444,A -85,B 0,C 180,E1 -1091.061,E2 -1091.061} C_VEL
LIN {X 0,Y 594.337,Z 124.447,A -85,B 0,C 180,E1 -1094.151,E2 -1094.151} C_VEL
LIN {X 0,Y 594.326,Z 124.448,A -85,B 0,C 180,E1 -1096.695,E2 -1096.695} C_VEL
LIN {X 0,Y 594.358,Z 124.454,A -85,B 0,C 180,E1 -1099.335,E2 -1099.335} C_VEL
LIN {X 0,Y 594.35,Z 124.451,A -85,B 0,C 180,E1 -1101.504,E2 -1101.504} C_VEL
LIN {X 0,Y 594.346,Z 124.445,A -85,B 0,C 180,E1 -1104.448,E2 -1104.448} C_VEL
LIN {X 0,Y 594.364,Z 124.448,A -85,B 0,C 180,E1 -1107.462,E2 -1107.462} C_VEL
LIN {X 0,Y 594.351,Z 124.445,A -85,B 0,C 180,E1 -1110.321,E2 -1110.321} C_VEL
LIN {X 0,Y 594.376,Z 124.451,A -85,B 0,C 180,E1 -1112.951,E2 -1112.951} C_VEL
LIN {X 0,Y 594.325,Z 124.451,A -85,B 0,C 180,E1 -1115.411,E2 -1115.411} C_VEL
LIN {X 0,Y 594.368,Z 124.442,A -85,B 0,C 180,E1 -1117.942,E2 -1117.942} C_VEL
LIN {X 0,Y 594.373,Z 124.452,A -85,B 0,C 180,E1 -1120.821,E2 -1120.821} C_VEL
LIN {X 0,Y 594.346,Z 124.445,A -85,B 0,C 180,E1 -1123.837,E2 -1123.837} C_VEL
LIN {X 0,Y 594.347,Z 124.455,A -85,B 0,C 180,E1 -1126.698,E2 -1126.698} C_VEL
LIN {X 0,Y 594.345,Z 124.445,A -85,B 0,C 180,E1 -1129.431,E2 -1129.431} C_VEL
LIN {X 0,Y 594.382,Z 124.448,A -85,B 0,C 180,E1 -1132.393,E2 -1132.393} C_VEL
LIN {X 0,Y 594.363,Z 124.443,A -85,B 0,C 180,E1 -1135.418,E2 -1135.418} C_VEL
LIN {X 0,Y 594.372,Z 124.452,A -85,B 0,C 180,E1 -1138.359,E2 -1138.359} C_VEL
LIN {X 0,Y 594.374,Z 124.442,A -85,B 0,C 180,E1 -1141.044,E2 -1141.044} C_VEL
LIN {X 0,Y 594.361,Z 124.444,A -85,B 0,C 180,E1 -1143.299,E2 -1143.299} C_VEL
LIN {X 0,Y 594.347,Z 124.448,A -85,B 0,C 180,E1 -1145.576,E2 -1145.576} C_VEL
LIN {X 0,Y 594.371,Z 124.547,A -85,B 0,C 180,E1 -1146.987,E2 -1146.987} C_VEL
LIN {X 0,Y 594.752,Z 129.042,A -85,B 0,C 180,E1 -1147.639,E2 -1147.639} C_VEL
LIN {X 0,Y 594.662,Z 149.466,A -85,B 0,C 180,E1 -1150.496,E2 -1150.496} C_VEL
LIN {X 0,Y 594.548,Z 171.472,A -85,B 0,C 180,E1 -1153.519,E2 -1153.519} C_VEL
LIN {X 0,Y 594.425,Z 193.478,A -85,B 0,C 180,E1 -1156.496,E2 -1156.496} C_VEL
LIN {X 0,Y 594.436,Z 194.611,A -85,B 0,C 180,E1 -1156.649,E2 -1156.649} C_VEL
LIN {X 0,Y 594.739,Z 198.7,A -85,B 0,C 180,E1 -1156.721,E2 -1156.721} C_VEL
LIN {X 0,Y 594.666,Z 302.935,A -85,B 0,C 180,E1 -1157.999,E2 -1157.999} C_VEL
LIN {X 0,Y 594.602,Z 316.211,A -85,B 0,C 180,E1 -1158.3,E2 -1158.3} C_VEL
LIN {X 0,Y 594.577,Z 328.486,A -85,B 0,C 180,E1 -1158.715,E2 -1158.715} C_VEL
LIN {X 0,Y 594.536,Z 340.627,A -85,B 0,C 180,E1 -1159.27,E2 -1159.27} C_VEL
LIN {X 0,Y 594.477,Z 352.198,A -85,B 0,C 180,E1 -1159.957,E2 -1159.957} C_VEL
LIN {X 0,Y 594.414,Z 362.595,A -85,B 0,C 180,E1 -1160.729,E2 -1160.729} C_VEL
LIN {X 0,Y 594.383,Z 371.11,A -85,B 0,C 180,E1 -1161.5,E2 -1161.5} C_VEL
LIN {X 0,Y 594.347,Z 378.959,A -85,B 0,C 180,E1 -1162.355,E2 -1162.355} C_VEL
LIN {X 0,Y 594.283,Z 386.813,A -85,B 0,C 180,E1 -1163.408,E2 -1163.408} C_VEL
LIN {X 0,Y 594.289,Z 393.679,A -85,B 0,C 180,E1 -1164.571,E2 -1164.571} C_VEL
LIN {X 0,Y 594.27,Z 398.371,A -85,B 0,C 180,E1 -1165.591,E2 -1165.591} C_VEL
LIN {X 0,Y 594.267,Z 401.956,A -85,B 0,C 180,E1 -1166.61,E2 -1166.61} C_VEL
LIN {X 0,Y 594.226,Z 403.808,A -85,B 0,C 180,E1 -1167.288,E2 -1167.288} C_VEL
LIN {X 0,Y 594.242,Z 405.2,A -85,B 0,C 180,E1 -1167.967,E2 -1167.967} C_VEL
LIN {X 0,Y 594.239,Z 406.784,A -85,B 0,C 180,E1 -1169.322,E2 -1169.322} C_VEL
LIN {X 0,Y 594.236,Z 407,A -85,B 0,C 180,E1 -1170,E2 -1170} C_VEL
LIN {X 0,Y 594.247,Z 406.185,A -85,B 0,C 180,E1 -1171.355,E2 -1171.355} C_VEL
LIN {X 0,Y 594.242,Z 405.201,A -85,B 0,C 180,E1 -1172.033,E2 -1172.033} C_VEL
LIN {X 0,Y 594.226,Z 403.81,A -85,B 0,C 180,E1 -1172.711,E2 -1172.711} C_VEL
LIN {X 0,Y 594.289,Z 400.896,A -85,B 0,C 180,E1 -1173.729,E2 -1173.729} C_VEL
LIN {X 0,Y 594.241,Z 396.95,A -85,B 0,C 180,E1 -1174.749,E2 -1174.749} C_VEL
LIN {X 0,Y 594.305,Z 390.878,A -85,B 0,C 180,E1 -1175.939,E2 -1175.939} C_VEL
LIN {X 0,Y 594.308,Z 384.237,A -85,B 0,C 180,E1 -1176.962,E2 -1176.962} C_VEL
LIN {X 0,Y 594.359,Z 375.99,A -85,B 0,C 180,E1 -1177.986,E2 -1177.986} C_VEL
LIN {X 0,Y 594.382,Z 367.538,A -85,B 0,C 180,E1 -1178.842,E2 -1178.842} C_VEL
LIN {X 0,Y 594.432,Z 357.095,A -85,B 0,C 180,E1 -1179.699,E2 -1179.699} C_VEL
LIN {X 0,Y 594.481,Z 346.759,A -85,B 0,C 180,E1 -1180.386,E2 -1180.386} C_VEL
LIN {X 0,Y 594.558,Z 335.727,A -85,B 0,C 180,E1 -1180.973,E2 -1180.973} C_VEL
LIN {X 0,Y 594.579,Z 323.713,A -85,B 0,C 180,E1 -1181.464,E2 -1181.464} C_VEL
LIN {X 0,Y 594.624,Z 310.351,A -85,B 0,C 180,E1 -1181.85,E2 -1181.85} C_VEL
LIN {X 0,Y 594.699,Z 297.086,A -85,B 0,C 180,E1 -1182.087,E2 -1182.087} C_VEL
LIN {X 0,Y 594.617,Z 196.262,A -85,B 0,C 180,E1 -1183.312,E2 -1183.312} C_VEL
LIN {X 0,Y 594.436,Z 194.613,A -85,B 0,C 180,E1 -1183.351,E2 -1183.351} C_VEL
LIN {X 0,Y 594.518,Z 172.769,A -85,B 0,C 180,E1 -1186.305,E2 -1186.305} C_VEL
LIN {X 0,Y 594.63,Z 152.408,A -85,B 0,C 180,E1 -1189.098,E2 -1189.098} C_VEL
LIN {X 0,Y 594.751,Z 131.345,A -85,B 0,C 180,E1 -1192.035,E2 -1192.035} C_VEL
LIN {X 0,Y 594.623,Z 126.021,A -85,B 0,C 180,E1 -1192.794,E2 -1192.794} C_VEL
LIN {X 0,Y 594.376,Z 124.447,A -85,B 0,C 180,E1 -1193.059,E2 -1193.059} C_VEL
LIN {X 0,Y 594.36,Z 124.449,A -85,B 0,C 180,E1 -1196.017,E2 -1196.017} C_VEL
LIN {X 0,Y 594.371,Z 124.444,A -85,B 0,C 180,E1 -1198.999,E2 -1198.999} C_VEL
LIN {X 0,Y 594.37,Z 124.451,A -85,B 0,C 180,E1 -1201.641,E2 -1201.641} C_VEL
LIN {X 0,Y 594.359,Z 124.444,A -85,B 0,C 180,E1 -1204.135,E2 -1204.135} C_VEL
LIN {X 0,Y 594.378,Z 124.447,A -85,B 0,C 180,E1 -1207.087,E2 -1207.087} C_VEL
LIN {X 0,Y 594.338,Z 124.449,A -85,B 0,C 180,E1 -1209.769,E2 -1209.769} C_VEL
LIN {X 0,Y 594.33,Z 124.448,A -85,B 0,C 180,E1 -1212.379,E2 -1212.379} C_VEL
LIN {X 0,Y 594.341,Z 124.455,A -85,B 0,C 180,E1 -1215.194,E2 -1215.194} C_VEL
LIN {X 0,Y 594.326,Z 124.449,A -85,B 0,C 180,E1 -1217.62,E2 -1217.62} C_VEL
LIN {X 0,Y 594.351,Z 124.446,A -85,B 0,C 180,E1 -1220.317,E2 -1220.317} C_VEL
LIN {X 0,Y 594.353,Z 124.454,A -85,B 0,C 180,E1 -1222.911,E2 -1222.911} C_VEL
LIN {X 0,Y 594.306,Z 124.45,A -85,B 0,C 180,E1 -1225.873,E2 -1225.873} C_VEL
LIN {X 0,Y 594.341,Z 124.456,A -85,B 0,C 180,E1 -1228.648,E2 -1228.648} C_VEL
LIN {X 0,Y 594.339,Z 124.449,A -85,B 0,C 180,E1 -1231.051,E2 -1231.051} C_VEL
LIN {X 0,Y 594.35,Z 124.444,A -85,B 0,C 180,E1 -1233.298,E2 -1233.298} C_VEL
LIN {X 0,Y 594.341,Z 124.454,A -85,B 0,C 180,E1 -1236.294,E2 -1236.294} C_VEL
LIN {X 0,Y 594.371,Z 124.442,A -85,B 0,C 180,E1 -1239.223,E2 -1239.223} C_VEL
LIN {X 0,Y 594.324,Z 124.455,A -85,B 0,C 180,E1 -1242.094,E2 -1242.094} C_VEL
LIN {X 0,Y 594.339,Z 124.455,A -85,B 0,C 180,E1 -1244.218,E2 -1244.218} C_VEL
LIN {X 0,Y 594.368,Z 124.448,A -85,B 0,C 180,E1 -1246.32,E2 -1246.32} C_VEL
LIN {X 0,Y 594.347,Z 124.445,A -85,B 0,C 180,E1 -1249.094,E2 -1249.094} C_VEL
LIN {X 0,Y 594.378,Z 124.45,A -85,B 0,C 180,E1 -1251.842,E2 -1251.842} C_VEL
LIN {X 0,Y 594.365,Z 124.443,A -85,B 0,C 180,E1 -1254.572,E2 -1254.572} C_VEL
LIN {X 0,Y 594.382,Z 124.443,A -85,B 0,C 180,E1 -1257.289,E2 -1257.289} C_VEL
LIN {X 0,Y 594.415,Z 124.441,A -85,B 0,C 180,E1 -1260,E2 -1260} C_VEL
LIN {X 0,Y 594.379,Z 124.441,A -85,B 0,C 180,E1 -1262.711,E2 -1262.711} C_VEL
LIN {X 0,Y 594.386,Z 124.45,A -85,B 0,C 180,E1 -1265.427,E2 -1265.427} C_VEL
LIN {X 0,Y 594.377,Z 124.442,A -85,B 0,C 180,E1 -1268.157,E2 -1268.157} C_VEL
LIN {X 0,Y 594.375,Z 124.447,A -85,B 0,C 180,E1 -1271.065,E2 -1271.065} C_VEL
LIN {X 0,Y 594.374,Z 124.444,A -85,B 0,C 180,E1 -1273.679,E2 -1273.679} C_VEL
LIN {X 0,Y 594.347,Z 124.45,A -85,B 0,C 180,E1 -1275.29,E2 -1275.29} C_VEL
LIN {X 0,Y 593.676,Z 124.531,A -85,B 0,C 180,E1 -1275.856,E2 -1275.856} C_VEL
LIN {X 0,Y 590.809,Z 124.89,A -85,B 0,C 180,E1 -1276.774,E2 -1276.774} C_VEL
LIN {X 0,Y 588.396,Z 125.189,A -85,B 0,C 180,E1 -1277.512,E2 -1277.512} C_VEL
LIN {X 0,Y 587.373,Z 125.314,A -85,B 0,C 180,E1 -1278.082,E2 -1278.082} C_VEL
LIN {X 0,Y 587.296,Z 125.323,A -85,B 0,C 180,E1 -1278.275,E2 -1278.275} C_VEL
LIN {X 0,Y 587.333,Z 125.327,A -85,B 0,C 180,E1 -1281.037,E2 -1281.037} C_VEL
LIN {X 0,Y 587.298,Z 125.324,A -85,B 0,C 180,E1 -1284.008,E2 -1284.008} C_VEL
LIN {X 0,Y 587.337,Z 125.321,A -85,B 0,C 180,E1 -1286.278,E2 -1286.278} C_VEL
LIN {X 0,Y 587.348,Z 125.32,A -85,B 0,C 180,E1 -1289.132,E2 -1289.132} C_VEL
LIN {X 0,Y 587.341,Z 125.318,A -85,B 0,C 180,E1 -1291.835,E2 -1291.835} C_VEL
LIN {X 0,Y 587.343,Z 125.325,A -85,B 0,C 180,E1 -1294.346,E2 -1294.346} C_VEL
LIN {X 0,Y 587.344,Z 125.318,A -85,B 0,C 180,E1 -1297.607,E2 -1297.607} C_VEL
LIN {X 0,Y 587.312,Z 125.33,A -85,B 0,C 180,E1 -1300.254,E2 -1300.254} C_VEL
LIN {X 0,Y 587.316,Z 125.322,A -85,B 0,C 180,E1 -1303.006,E2 -1303.006} C_VEL
LIN {X 0,Y 587.323,Z 125.329,A -85,B 0,C 180,E1 -1306.049,E2 -1306.049} C_VEL
LIN {X 0,Y 587.336,Z 125.32,A -85,B 0,C 180,E1 -1308.924,E2 -1308.924} C_VEL
LIN {X 0,Y 587.371,Z 125.466,A -85,B 0,C 180,E1 -1311.113,E2 -1311.113} C_VEL
LIN {X 0,Y 587.428,Z 138.83,A -85,B 0,C 180,E1 -1313.488,E2 -1313.488} C_VEL
LIN {X 0,Y 587.34,Z 155.452,A -85,B 0,C 180,E1 -1316.398,E2 -1316.398} C_VEL
LIN {X 0,Y 587.378,Z 156.723,A -85,B 0,C 180,E1 -1316.572,E2 -1316.572} C_VEL
LIN {X 0,Y 587.865,Z 161.107,A -85,B 0,C 180,E1 -1316.637,E2 -1316.637} C_VEL
LIN {X 0,Y 587.726,Z 263.644,A -85,B 0,C 180,E1 -1317.913,E2 -1317.913} C_VEL
LIN {X 0,Y 587.672,Z 277.263,A -85,B 0,C 180,E1 -1318.236,E2 -1318.236} C_VEL
LIN {X 0,Y 587.579,Z 290.314,A -85,B 0,C 180,E1 -1318.698,E2 -1318.698} C_VEL
LIN {X 0,Y 587.483,Z 302.554,A -85,B 0,C 180,E1 -1319.291,E2 -1319.291} C_VEL
LIN {X 0,Y 587.436,Z 314.442,A -85,B 0,C 180,E1 -1320.034,E2 -1320.034} C_VEL
LIN {X 0,Y 587.378,Z 324.903,A -85,B 0,C 180,E1 -1320.861,E2 -1320.861} C_VEL
LIN {X 0,Y 587.307,Z 334.44,A -85,B 0,C 180,E1 -1321.792,E2 -1321.792} C_VEL
LIN {X 0,Y 587.266,Z 342.513,A -85,B 0,C 180,E1 -1322.759,E2 -1322.759} C_VEL
LIN {X 0,Y 587.215,Z 349.781,A -85,B 0,C 180,E1 -1323.847,E2 -1323.847} C_VEL
LIN {X 0,Y 587.194,Z 355.184,A -85,B 0,C 180,E1 -1324.856,E2 -1324.856} C_VEL
LIN {X 0,Y 587.177,Z 359.893,A -85,B 0,C 180,E1 -1325.987,E2 -1325.987} C_VEL
LIN {X 0,Y 587.144,Z 363.478,A -85,B 0,C 180,E1 -1327.171,E2 -1327.171} C_VEL
LIN {X 0,Y 587.141,Z 365.574,A -85,B 0,C 180,E1 -1328.219,E2 -1328.219} C_VEL
LIN {X 0,Y 587.144,Z 366.544,A -85,B 0,C 180,E1 -1329.009,E2 -1329.009} C_VEL
LIN {X 0,Y 587.121,Z 366.925,A -85,B 0,C 180,E1 -1329.688,E2 -1329.688} C_VEL
LIN {X 0,Y 587.148,Z 366.59,A -85,B 0,C 180,E1 -1331.014,E2 -1331.014} C_VEL
LIN {X 0,Y 587.127,Z 365.581,A -85,B 0,C 180,E1 -1331.867,E2 -1331.867} C_VEL
LIN {X 0,Y 587.134,Z 364.245,A -85,B 0,C 180,E1 -1332.587,E2 -1332.587} C_VEL
LIN {X 0,Y 587.158,Z 361.38,A -85,B 0,C 180,E1 -1333.663,E2 -1333.663} C_VEL
LIN {X 0,Y 587.184,Z 357.438,A -85,B 0,C 180,E1 -1334.733,E2 -1334.733} C_VEL
LIN {X 0,Y 587.229,Z 351.803,A -85,B 0,C 180,E1 -1335.895,E2 -1335.895} C_VEL
LIN {X 0,Y 587.24,Z 344.656,A -85,B 0,C 180,E1 -1337.033,E2 -1337.033} C_VEL
LIN {X 0,Y 587.332,Z 336.332,A -85,B 0,C 180,E1 -1338.088,E2 -1338.088} C_VEL
LIN {X 0,Y 587.348,Z 327.874,A -85,B 0,C 180,E1 -1338.963,E2 -1338.963} C_VEL
LIN {X 0,Y 587.445,Z 317.427,A -85,B 0,C 180,E1 -1339.836,E2 -1339.836} C_VEL
LIN {X 0,Y 587.519,Z 305.708,A -85,B 0,C 180,E1 -1340.62,E2 -1340.62} C_VEL
LIN {X 0,Y 587.569,Z 294.048,A -85,B 0,C 180,E1 -1341.228,E2 -1341.228} C_VEL
LIN {X 0,Y 587.603,Z 282.008,A -85,B 0,C 180,E1 -1341.705,E2 -1341.705} C_VEL
LIN {X 0,Y 587.66,Z 268.875,A -85,B 0,C 180,E1 -1342.073,E2 -1342.073} C_VEL
LIN {X 0,Y 587.707,Z 256.099,A -85,B 0,C 180,E1 -1342.29,E2 -1342.29} C_VEL
LIN {X 0,Y 587.726,Z 159.076,A -85,B 0,C 180,E1 -1343.481,E2 -1343.481} C_VEL
LIN {X 0,Y 587.309,Z 156.295,A -85,B 0,C 180,E1 -1343.546,E2 -1343.546} C_VEL
LIN {X 0,Y 587.403,Z 140.96,A -85,B 0,C 180,E1 -1346.227,E2 -1346.227} C_VEL
LIN {X 0,Y 587.458,Z 127.396,A -85,B 0,C 180,E1 -1348.629,E2 -1348.629} C_VEL
LIN {X 0,Y 587.278,Z 125.33,A -85,B 0,C 180,E1 -1349.014,E2 -1349.014} C_VEL
LIN {X 0,Y 587.273,Z 125.328,A -85,B 0,C 180,E1 -1350.686,E2 -1350.686} C_VEL
LIN {X 0,Y 587.329,Z 125.321,A -85,B 0,C 180,E1 -1352.744,E2 -1352.744} C_VEL
LIN {X 0,Y 587.324,Z 125.323,A -85,B 0,C 180,E1 -1355.493,E2 -1355.493} C_VEL
LIN {X 0,Y 587.321,Z 125.324,A -85,B 0,C 180,E1 -1358.256,E2 -1358.256} C_VEL
LIN {X 0,Y 587.292,Z 125.325,A -85,B 0,C 180,E1 -1361.107,E2 -1361.107} C_VEL
LIN {X 0,Y 587.326,Z 125.328,A -85,B 0,C 180,E1 -1363.847,E2 -1363.847} C_VEL
LIN {X 0,Y 587.288,Z 125.324,A -85,B 0,C 180,E1 -1366.796,E2 -1366.796} C_VEL
LIN {X 0,Y 587.278,Z 125.336,A -85,B 0,C 180,E1 -1369.578,E2 -1369.578} C_VEL
LIN {X 0,Y 587.285,Z 125.331,A -85,B 0,C 180,E1 -1371.776,E2 -1371.776} C_VEL
LIN {X 0,Y 587.285,Z 125.325,A -85,B 0,C 180,E1 -1374.762,E2 -1374.762} C_VEL
LIN {X 0,Y 587.291,Z 125.329,A -85,B 0,C 180,E1 -1377.683,E2 -1377.683} C_VEL
LIN {X 0,Y 587.282,Z 125.325,A -85,B 0,C 180,E1 -1380.502,E2 -1380.502} C_VEL
LIN {X 0,Y 587.297,Z 125.331,A -85,B 0,C 180,E1 -1383.4,E2 -1383.4} C_VEL
LIN {X 0,Y 587.249,Z 125.33,A -85,B 0,C 180,E1 -1385.903,E2 -1385.903} C_VEL
LIN {X 0,Y 587.286,Z 125.326,A -85,B 0,C 180,E1 -1388.483,E2 -1388.483} C_VEL
LIN {X 0,Y 587.296,Z 125.332,A -85,B 0,C 180,E1 -1391.161,E2 -1391.161} C_VEL
LIN {X 0,Y 587.3,Z 125.323,A -85,B 0,C 180,E1 -1394.111,E2 -1394.111} C_VEL
LIN {X 0,Y 587.279,Z 125.334,A -85,B 0,C 180,E1 -1396.991,E2 -1396.991} C_VEL
LIN {X 0,Y 587.289,Z 125.324,A -85,B 0,C 180,E1 -1399.744,E2 -1399.744} C_VEL
LIN {X 0,Y 587.328,Z 125.323,A -85,B 0,C 180,E1 -1402.392,E2 -1402.392} C_VEL
LIN {X 0,Y 587.302,Z 125.322,A -85,B 0,C 180,E1 -1405.66,E2 -1405.66} C_VEL
LIN {X 0,Y 587.299,Z 125.326,A -85,B 0,C 180,E1 -1408.229,E2 -1408.229} C_VEL
LIN {X 0,Y 587.299,Z 125.328,A -85,B 0,C 180,E1 -1410.877,E2 -1410.877} C_VEL
LIN {X 0,Y 587.305,Z 125.323,A -85,B 0,C 180,E1 -1413.831,E2 -1413.831} C_VEL
LIN {X 0,Y 587.287,Z 125.329,A -85,B 0,C 180,E1 -1416.74,E2 -1416.74} C_VEL
LIN {X 0,Y 587.298,Z 125.324,A -85,B 0,C 180,E1 -1419.694,E2 -1419.694} C_VEL
LIN {X 0,Y 587.271,Z 125.331,A -85,B 0,C 180,E1 -1422.592,E2 -1422.592} C_VEL
LIN {X 0,Y 587.313,Z 125.322,A -85,B 0,C 180,E1 -1425.446,E2 -1425.446} C_VEL
LIN {X 0,Y 587.314,Z 125.329,A -85,B 0,C 180,E1 -1428.263,E2 -1428.263} C_VEL
LIN {X 0,Y 587.279,Z 125.325,A -85,B 0,C 180,E1 -1431.05,E2 -1431.05} C_VEL
LIN {X 0,Y 587.311,Z 125.328,A -85,B 0,C 180,E1 -1433.818,E2 -1433.818} C_VEL
LIN {X 0,Y 587.304,Z 125.332,A -85,B 0,C 180,E1 -1435.883,E2 -1435.883} C_VEL
LIN {X 0,Y 587.371,Z 125.323,A -85,B 0,C 180,E1 -1437.943,E2 -1437.943} C_VEL
LIN {X 0,Y 587.383,Z 125.32,A -85,B 0,C 180,E1 -1440,E2 -1440} C_VEL
LIN {X 0,Y 587.333,Z 125.318,A -85,B 0,C 180,E1 -1442.744,E2 -1442.744} C_VEL
LIN {X 0,Y 587.336,Z 125.325,A -85,B 0,C 180,E1 -1445.494,E2 -1445.494} C_VEL
LIN {X 0,Y 587.329,Z 125.32,A -85,B 0,C 180,E1 -1448.256,E2 -1448.256} C_VEL
LIN {X 0,Y 587.337,Z 125.321,A -85,B 0,C 180,E1 -1451.125,E2 -1451.125} C_VEL
LIN {X 0,Y 587.307,Z 125.322,A -85,B 0,C 180,E1 -1454.235,E2 -1454.235} C_VEL
LIN {X 0,Y 587.298,Z 125.324,A -85,B 0,C 180,E1 -1456.796,E2 -1456.796} C_VEL
LIN {X 0,Y 587.3,Z 125.329,A -85,B 0,C 180,E1 -1459.577,E2 -1459.577} C_VEL
LIN {X 0,Y 587.299,Z 125.326,A -85,B 0,C 180,E1 -1461.776,E2 -1461.776} C_VEL
LIN {X 0,Y 587.302,Z 125.325,A -85,B 0,C 180,E1 -1464.761,E2 -1464.761} C_VEL
LIN {X 0,Y 587.301,Z 125.325,A -85,B 0,C 180,E1 -1467.682,E2 -1467.682} C_VEL
LIN {X 0,Y 587.31,Z 125.323,A -85,B 0,C 180,E1 -1470.504,E2 -1470.504} C_VEL
LIN {X 0,Y 587.324,Z 125.323,A -85,B 0,C 180,E1 -1473.398,E2 -1473.398} C_VEL
LIN {X 0,Y 587.279,Z 125.325,A -85,B 0,C 180,E1 -1475.901,E2 -1475.901} C_VEL
LIN {X 0,Y 587.315,Z 125.325,A -85,B 0,C 180,E1 -1478.481,E2 -1478.481} C_VEL
LIN {X 0,Y 587.333,Z 125.323,A -85,B 0,C 180,E1 -1481.158,E2 -1481.158} C_VEL
LIN {X 0,Y 587.306,Z 125.323,A -85,B 0,C 180,E1 -1484.111,E2 -1484.111} C_VEL
LIN {X 0,Y 587.29,Z 125.329,A -85,B 0,C 180,E1 -1486.991,E2 -1486.991} C_VEL
LIN {X 0,Y 587.297,Z 125.323,A -85,B 0,C 180,E1 -1489.744,E2 -1489.744} C_VEL
LIN {X 0,Y 587.336,Z 125.326,A -85,B 0,C 180,E1 -1492.391,E2 -1492.391} C_VEL
LIN {X 0,Y 587.332,Z 125.319,A -85,B 0,C 180,E1 -1495.655,E2 -1495.655} C_VEL
LIN {X 0,Y 587.335,Z 125.326,A -85,B 0,C 180,E1 -1498.23,E2 -1498.23} C_VEL
LIN {X 0,Y 587.343,Z 125.32,A -85,B 0,C 180,E1 -1500.868,E2 -1500.868} C_VEL
LIN {X 0,Y 587.311,Z 125.326,A -85,B 0,C 180,E1 -1503.829,E2 -1503.829} C_VEL
LIN {X 0,Y 587.32,Z 125.426,A -85,B 0,C 180,E1 -1506.847,E2 -1506.847} C_VEL
LIN {X 0,Y 587.833,Z 129.961,A -85,B 0,C 180,E1 -1507.506,E2 -1507.506} C_VEL
LIN {X 0,Y 587.741,Z 149.466,A -85,B 0,C 180,E1 -1510.257,E2 -1510.257} C_VEL
LIN {X 0,Y 587.525,Z 170.129,A -85,B 0,C 180,E1 -1513.13,E2 -1513.13} C_VEL
LIN {X 0,Y 587.451,Z 189.886,A -85,B 0,C 180,E1 -1515.843,E2 -1515.843} C_VEL
LIN {X 0,Y 587.381,Z 194.611,A -85,B 0,C 180,E1 -1516.485,E2 -1516.485} C_VEL
LIN {X 0,Y 587.838,Z 198.7,A -85,B 0,C 180,E1 -1516.562,E2 -1516.562} C_VEL
LIN {X 0,Y 587.725,Z 302.935,A -85,B 0,C 180,E1 -1517.855,E2 -1517.855} C_VEL
LIN {X 0,Y 587.668,Z 316.212,A -85,B 0,C 180,E1 -1518.16,E2 -1518.16} C_VEL
LIN {X 0,Y 587.607,Z 328.638,A -85,B 0,C 180,E1 -1518.585,E2 -1518.585} C_VEL
LIN {X 0,Y 587.558,Z 340.626,A -85,B 0,C 180,E1 -1519.141,E2 -1519.141} C_VEL
LIN {X 0,Y 587.464,Z 352.2,A -85,B 0,C 180,E1 -1519.836,E2 -1519.836} C_VEL
LIN {X 0,Y 587.366,Z 362.597,A -85,B 0,C 180,E1 -1520.617,E2 -1520.617} C_VEL
LIN {X 0,Y 587.322,Z 371.11,A -85,B 0,C 180,E1 -1521.397,E2 -1521.397} C_VEL
LIN {X 0,Y 587.274,Z 378.959,A -85,B 0,C 180,E1 -1522.263,E2 -1522.263} C_VEL
LIN {X 0,Y 587.23,Z 385.468,A -85,B 0,C 180,E1 -1523.126,E2 -1523.126} C_VEL
LIN {X 0,Y 587.237,Z 391.866,A -85,B 0,C 180,E1 -1524.161,E2 -1524.161} C_VEL
LIN {X 0,Y 587.147,Z 396.949,A -85,B 0,C 180,E1 -1525.193,E2 -1525.193} C_VEL
LIN {X 0,Y 587.213,Z 400.895,A -85,B 0,C 180,E1 -1526.226,E2 -1526.226} C_VEL
LIN {X 0,Y 587.132,Z 403.808,A -85,B 0,C 180,E1 -1527.255,E2 -1527.255} C_VEL
LIN {X 0,Y 587.141,Z 405.199,A -85,B 0,C 180,E1 -1527.942,E2 -1527.942} C_VEL
LIN {X 0,Y 587.14,Z 406.784,A -85,B 0,C 180,E1 -1529.314,E2 -1529.314} C_VEL
LIN {X 0,Y 587.137,Z 407,A -85,B 0,C 180,E1 -1530,E2 -1530} C_VEL
LIN {X 0,Y 587.147,Z 406.186,A -85,B 0,C 180,E1 -1531.372,E2 -1531.372} C_VEL
LIN {X 0,Y 587.141,Z 405.201,A -85,B 0,C 180,E1 -1532.058,E2 -1532.058} C_VEL
LIN {X 0,Y 587.132,Z 403.81,A -85,B 0,C 180,E1 -1532.744,E2 -1532.744} C_VEL
LIN {X 0,Y 587.213,Z 400.896,A -85,B 0,C 180,E1 -1533.774,E2 -1533.774} C_VEL
LIN {X 0,Y 587.147,Z 396.95,A -85,B 0,C 180,E1 -1534.806,E2 -1534.806} C_VEL
LIN {X 0,Y 587.218,Z 390.878,A -85,B 0,C 180,E1 -1536.011,E2 -1536.011} C_VEL
LIN {X 0,Y 587.245,Z 384.238,A -85,B 0,C 180,E1 -1537.046,E2 -1537.046} C_VEL
LIN {X 0,Y 587.299,Z 375.991,A -85,B 0,C 180,E1 -1538.083,E2 -1538.083} C_VEL
LIN {X 0,Y 587.343,Z 367.539,A -85,B 0,C 180,E1 -1538.949,E2 -1538.949} C_VEL
LIN {X 0,Y 587.419,Z 357.097,A -85,B 0,C 180,E1 -1539.816,E2 -1539.816} C_VEL
LIN {X 0,Y 587.497,Z 346.757,A -85,B 0,C 180,E1 -1540.511,E2 -1540.511} C_VEL
LIN {X 0,Y 587.561,Z 334.819,A -85,B 0,C 180,E1 -1541.149,E2 -1541.149} C_VEL
LIN {X 0,Y 587.629,Z 322.6,A -85,B 0,C 180,E1 -1541.639,E2 -1541.639} C_VEL
LIN {X 0,Y 587.704,Z 309.436,A -85,B 0,C 180,E1 -1542.014,E2 -1542.014} C_VEL
LIN {X 0,Y 587.785,Z 297.086,A -85,B 0,C 180,E1 -1542.231,E2 -1542.231} C_VEL
LIN {X 0,Y 587.709,Z 196.708,A -85,B 0,C 180,E1 -1543.465,E2 -1543.465} C_VEL
LIN {X 0,Y 587.381,Z 194.613,A -85,B 0,C 180,E1 -1543.514,E2 -1543.514} C_VEL
LIN {X 0,Y 587.542,Z 174.063,A -85,B 0,C 180,E1 -1546.326,E2 -1546.326} C_VEL
LIN {X 0,Y 587.669,Z 153.85,A -85,B 0,C 180,E1 -1549.131,E2 -1549.131} C_VEL
LIN {X 0,Y 587.824,Z 135.225,A -85,B 0,C 180,E1 -1551.755,E2 -1551.755} C_VEL
LIN {X 0,Y 587.609,Z 126.861,A -85,B 0,C 180,E1 -1552.935,E2 -1552.935} C_VEL
LIN {X 0,Y 587.314,Z 125.328,A -85,B 0,C 180,E1 -1553.18,E2 -1553.18} C_VEL
LIN {X 0,Y 587.31,Z 125.326,A -85,B 0,C 180,E1 -1556.17,E2 -1556.17} C_VEL
LIN {X 0,Y 587.342,Z 125.321,A -85,B 0,C 180,E1 -1559.131,E2 -1559.131} C_VEL
LIN {X 0,Y 587.316,Z 125.326,A -85,B 0,C 180,E1 -1561.831,E2 -1561.831} C_VEL
LIN {X 0,Y 587.328,Z 125.319,A -85,B 0,C 180,E1 -1564.344,E2 -1564.344} C_VEL
LIN {X 0,Y 587.333,Z 125.325,A -85,B 0,C 180,E1 -1567.609,E2 -1567.609} C_VEL
LIN {X 0,Y 587.293,Z 125.324,A -85,B 0,C 180,E1 -1570.256,E2 -1570.256} C_VEL
LIN {X 0,Y 587.288,Z 125.334,A -85,B 0,C 180,E1 -1573.115,E2 -1573.115} C_VEL
LIN {X 0,Y 587.299,Z 125.323,A -85,B 0,C 180,E1 -1576.047,E2 -1576.047} C_VEL
LIN {X 0,Y 587.302,Z 125.332,A -85,B 0,C 180,E1 -1578.929,E2 -1578.929} C_VEL
LIN {X 0,Y 587.272,Z 125.328,A -85,B 0,C 180,E1 -1581.516,E2 -1581.516} C_VEL
LIN {X 0,Y 587.252,Z 125.33,A -85,B 0,C 180,E1 -1584.097,E2 -1584.097} C_VEL
LIN {X 0,Y 587.281,Z 125.332,A -85,B 0,C 180,E1 -1586.898,E2 -1586.898} C_VEL
LIN {X 0,Y 587.287,Z 125.324,A -85,B 0,C 180,E1 -1589.499,E2 -1589.499} C_VEL
LIN {X 0,Y 587.297,Z 125.329,A -85,B 0,C 180,E1 -1592.318,E2 -1592.318} C_VEL
LIN {X 0,Y 587.292,Z 125.324,A -85,B 0,C 180,E1 -1595.238,E2 -1595.238} C_VEL
LIN {X 0,Y 587.293,Z 125.331,A -85,B 0,C 180,E1 -1598.224,E2 -1598.224} C_VEL
LIN {X 0,Y 587.292,Z 125.324,A -85,B 0,C 180,E1 -1601.149,E2 -1601.149} C_VEL
LIN {X 0,Y 587.289,Z 125.332,A -85,B 0,C 180,E1 -1604.023,E2 -1604.023} C_VEL
LIN {X 0,Y 587.345,Z 125.326,A -85,B 0,C 180,E1 -1606.154,E2 -1606.154} C_VEL
LIN {X 0,Y 587.322,Z 125.32,A -85,B 0,C 180,E1 -1608.962,E2 -1608.962} C_VEL
LIN {X 0,Y 587.337,Z 125.325,A -85,B 0,C 180,E1 -1611.744,E2 -1611.744} C_VEL
LIN {X 0,Y 587.334,Z 125.319,A -85,B 0,C 180,E1 -1614.506,E2 -1614.506} C_VEL
LIN {X 0,Y 587.348,Z 125.318,A -85,B 0,C 180,E1 -1617.256,E2 -1617.256} C_VEL
LIN {X 0,Y 587.384,Z 125.316,A -85,B 0,C 180,E1 -1620,E2 -1620} C_VEL
LIN {X 0,Y 587.349,Z 125.317,A -85,B 0,C 180,E1 -1622.743,E2 -1622.743} C_VEL
LIN {X 0,Y 587.351,Z 125.325,A -85,B 0,C 180,E1 -1625.493,E2 -1625.493} C_VEL
LIN {X 0,Y 587.337,Z 125.318,A -85,B 0,C 180,E1 -1628.255,E2 -1628.255} C_VEL
LIN {X 0,Y 587.352,Z 125.323,A -85,B 0,C 180,E1 -1631.133,E2 -1631.133} C_VEL
LIN {X 0,Y 587.334,Z 125.318,A -85,B 0,C 180,E1 -1634.247,E2 -1634.247} C_VEL
LIN {X 0,Y 587.333,Z 125.324,A -85,B 0,C 180,E1 -1636.808,E2 -1636.808} C_VEL
LIN {X 0,Y 587.296,Z 125.323,A -85,B 0,C 180,E1 -1638.275,E2 -1638.275} C_VEL
LIN {X 0,Y 586.659,Z 125.41,A -85,B 0,C 180,E1 -1638.847,E2 -1638.847} C_VEL
LIN {X 0,Y 583.852,Z 125.762,A -85,B 0,C 180,E1 -1639.776,E2 -1639.776} C_VEL
LIN {X 0,Y 581.448,Z 126.062,A -85,B 0,C 180,E1 -1640.523,E2 -1640.523} C_VEL
LIN {X 0,Y 580.387,Z 126.191,A -85,B 0,C 180,E1 -1641.099,E2 -1641.099} C_VEL
LIN {X 0,Y 580.286,Z 126.201,A -85,B 0,C 180,E1 -1641.294,E2 -1641.294} C_VEL
LIN {X 0,Y 580.257,Z 126.202,A -85,B 0,C 180,E1 -1643.558,E2 -1643.558} C_VEL
LIN {X 0,Y 580.29,Z 126.199,A -85,B 0,C 180,E1 -1646.333,E2 -1646.333} C_VEL
LIN {X 0,Y 580.297,Z 126.197,A -85,B 0,C 180,E1 -1649.308,E2 -1649.308} C_VEL
LIN {X 0,Y 580.297,Z 126.199,A -85,B 0,C 180,E1 -1652.2,E2 -1652.2} C_VEL
LIN {X 0,Y 580.288,Z 126.204,A -85,B 0,C 180,E1 -1654.696,E2 -1654.696} C_VEL
LIN {X 0,Y 580.298,Z 126.196,A -85,B 0,C 180,E1 -1657.268,E2 -1657.268} C_VEL
LIN {X 0,Y 580.291,Z 126.205,A -85,B 0,C 180,E1 -1660.27,E2 -1660.27} C_VEL
LIN {X 0,Y 580.278,Z 126.202,A -85,B 0,C 180,E1 -1662.706,E2 -1662.706} C_VEL
LIN {X 0,Y 580.269,Z 126.202,A -85,B 0,C 180,E1 -1665.609,E2 -1665.609} C_VEL
LIN {X 0,Y 580.288,Z 126.205,A -85,B 0,C 180,E1 -1668.232,E2 -1668.232} C_VEL
LIN {X 0,Y 580.319,Z 126.285,A -85,B 0,C 180,E1 -1671.024,E2 -1671.024} C_VEL
LIN {X 0,Y 580.451,Z 135.81,A -85,B 0,C 180,E1 -1672.743,E2 -1672.743} C_VEL
LIN {X 0,Y 580.333,Z 151.955,A -85,B 0,C 180,E1 -1675.613,E2 -1675.613} C_VEL
LIN {X 0,Y 580.308,Z 156.481,A -85,B 0,C 180,E1 -1676.402,E2 -1676.402} C_VEL
LIN {X 0,Y 580.962,Z 161.701,A -85,B 0,C 180,E1 -1676.482,E2 -1676.482} C_VEL
LIN {X 0,Y 580.785,Z 263.608,A -85,B 0,C 180,E1 -1677.766,E2 -1677.766} C_VEL
LIN {X 0,Y 580.738,Z 276.91,A -85,B 0,C 180,E1 -1678.082,E2 -1678.082} C_VEL
LIN {X 0,Y 580.638,Z 289.722,A -85,B 0,C 180,E1 -1678.535,E2 -1678.535} C_VEL
LIN {X 0,Y 580.532,Z 301.088,A -85,B 0,C 180,E1 -1679.079,E2 -1679.079} C_VEL
LIN {X 0,Y 580.397,Z 313.315,A -85,B 0,C 180,E1 -1679.833,E2 -1679.833} C_VEL
LIN {X 0,Y 580.344,Z 324.164,A -85,B 0,C 180,E1 -1680.682,E2 -1680.682} C_VEL
LIN {X 0,Y 580.277,Z 333.745,A -85,B 0,C 180,E1 -1681.616,E2 -1681.616} C_VEL
LIN {X 0,Y 580.205,Z 341.928,A -85,B 0,C 180,E1 -1682.594,E2 -1682.594} C_VEL
LIN {X 0,Y 580.136,Z 349.351,A -85,B 0,C 180,E1 -1683.696,E2 -1683.696} C_VEL
LIN {X 0,Y 580.114,Z 355.733,A -85,B 0,C 180,E1 -1684.911,E2 -1684.911} C_VEL
LIN {X 0,Y 580.088,Z 360.311,A -85,B 0,C 180,E1 -1686.055,E2 -1686.055} C_VEL
LIN {X 0,Y 580.071,Z 363.613,A -85,B 0,C 180,E1 -1687.188,E2 -1687.188} C_VEL
LIN {X 0,Y 580.032,Z 365.16,A -85,B 0,C 180,E1 -1687.938,E2 -1687.938} C_VEL
LIN {X 0,Y 580.04,Z 366.46,A -85,B 0,C 180,E1 -1688.9,E2 -1688.9} C_VEL
LIN {X 0,Y 580.02,Z 366.979,A -85,B 0,C 180,E1 -1690.168,E2 -1690.168} C_VEL
LIN {X 0,Y 580.062,Z 366.666,A -85,B 0,C 180,E1 -1690.915,E2 -1690.915} C_VEL
LIN {X 0,Y 580.035,Z 365.951,A -85,B 0,C 180,E1 -1691.637,E2 -1691.637} C_VEL
LIN {X 0,Y 580.043,Z 364.763,A -85,B 0,C 180,E1 -1692.368,E2 -1692.368} C_VEL
LIN {X 0,Y 580.041,Z 362.918,A -85,B 0,C 180,E1 -1693.173,E2 -1693.173} C_VEL
LIN {X 0,Y 580.077,Z 359.794,A -85,B 0,C 180,E1 -1694.181,E2 -1694.181} C_VEL
LIN {X 0,Y 580.125,Z 355.35,A -85,B 0,C 180,E1 -1695.262,E2 -1695.262} C_VEL
LIN {X 0,Y 580.117,Z 349.69,A -85,B 0,C 180,E1 -1696.335,E2 -1696.335} C_VEL
LIN {X 0,Y 580.208,Z 342.611,A -85,B 0,C 180,E1 -1697.407,E2 -1697.407} C_VEL
LIN {X 0,Y 580.269,Z 333.757,A -85,B 0,C 180,E1 -1698.473,E2 -1698.473} C_VEL
LIN {X 0,Y 580.323,Z 324.6,A -85,B 0,C 180,E1 -1699.369,E2 -1699.369} C_VEL
LIN {X 0,Y 580.405,Z 314.818,A -85,B 0,C 180,E1 -1700.152,E2 -1700.152} C_VEL
LIN {X 0,Y 580.531,Z 303.835,A -85,B 0,C 180,E1 -1700.857,E2 -1700.857} C_VEL
LIN {X 0,Y 580.644,Z 291.584,A -85,B 0,C 180,E1 -1701.473,E2 -1701.473} C_VEL
LIN {X 0,Y 580.689,Z 278.732,A -85,B 0,C 180,E1 -1701.956,E2 -1701.956} C_VEL
LIN {X 0,Y 580.773,Z 265.65,A -85,B 0,C 180,E1 -1702.285,E2 -1702.285} C_VEL
LIN {X 0,Y 580.853,Z 247.102,A -85,B 0,C 180,E1 -1702.549,E2 -1702.549} C_VEL
LIN {X 0,Y 580.819,Z 159.765,A -85,B 0,C 180,E1 -1703.635,E2 -1703.635} C_VEL
LIN {X 0,Y 580.244,Z 156.419,A -85,B 0,C 180,E1 -1703.692,E2 -1703.692} C_VEL
LIN {X 0,Y 580.38,Z 142.345,A -85,B 0,C 180,E1 -1706.181,E2 -1706.181} C_VEL
LIN {X 0,Y 580.455,Z 128.775,A -85,B 0,C 180,E1 -1708.613,E2 -1708.613} C_VEL
LIN {X 0,Y 580.234,Z 126.208,A -85,B 0,C 180,E1 -1709.089,E2 -1709.089} C_VEL
LIN {X 0,Y 580.228,Z 126.206,A -85,B 0,C 180,E1 -1710.694,E2 -1710.694} C_VEL
LIN {X 0,Y 580.297,Z 126.197,A -85,B 0,C 180,E1 -1712.777,E2 -1712.777} C_VEL
LIN {X 0,Y 580.293,Z 126.199,A -85,B 0,C 180,E1 -1715.56,E2 -1715.56} C_VEL
LIN {X 0,Y 580.287,Z 126.199,A -85,B 0,C 180,E1 -1718.357,E2 -1718.357} C_VEL
LIN {X 0,Y 580.263,Z 126.201,A -85,B 0,C 180,E1 -1721.174,E2 -1721.174} C_VEL
LIN {X 0,Y 580.275,Z 126.199,A -85,B 0,C 180,E1 -1724.324,E2 -1724.324} C_VEL
LIN {X 0,Y 580.246,Z 126.202,A -85,B 0,C 180,E1 -1726.9,E2 -1726.9} C_VEL
LIN {X 0,Y 580.24,Z 126.208,A -85,B 0,C 180,E1 -1729.825,E2 -1729.825} C_VEL
LIN {X 0,Y 580.221,Z 126.207,A -85,B 0,C 180,E1 -1732.055,E2 -1732.055} C_VEL
LIN {X 0,Y 580.239,Z 126.203,A -85,B 0,C 180,E1 -1734.713,E2 -1734.713} C_VEL
LIN {X 0,Y 580.239,Z 126.213,A -85,B 0,C 180,E1 -1737.405,E2 -1737.405} C_VEL
LIN {X 0,Y 580.241,Z 126.205,A -85,B 0,C 180,E1 -1739.776,E2 -1739.776} C_VEL
LIN {X 0,Y 580.264,Z 126.199,A -85,B 0,C 180,E1 -1742.203,E2 -1742.203} C_VEL
LIN {X 0,Y 580.259,Z 126.202,A -85,B 0,C 180,E1 -1744.699,E2 -1744.699} C_VEL
LIN {X 0,Y 580.263,Z 126.207,A -85,B 0,C 180,E1 -1747.272,E2 -1747.272} C_VEL
LIN {X 0,Y 580.269,Z 126.199,A -85,B 0,C 180,E1 -1750.268,E2 -1750.268} C_VEL
LIN {X 0,Y 580.228,Z 126.207,A -85,B 0,C 180,E1 -1753.386,E2 -1753.386} C_VEL
LIN {X 0,Y 580.249,Z 126.202,A -85,B 0,C 180,E1 -1755.612,E2 -1755.612} C_VEL
LIN {X 0,Y 580.235,Z 126.204,A -85,B 0,C 180,E1 -1758.228,E2 -1758.228} C_VEL
LIN {X 0,Y 580.257,Z 126.207,A -85,B 0,C 180,E1 -1760.964,E2 -1760.964} C_VEL
LIN {X 0,Y 580.234,Z 126.203,A -85,B 0,C 180,E1 -1763.594,E2 -1763.594} C_VEL
LIN {X 0,Y 580.252,Z 126.203,A -85,B 0,C 180,E1 -1766.142,E2 -1766.142} C_VEL
LIN {X 0,Y 580.239,Z 126.213,A -85,B 0,C 180,E1 -1768.613,E2 -1768.613} C_VEL
LIN {X 0,Y 580.244,Z 126.205,A -85,B 0,C 180,E1 -1771.022,E2 -1771.022} C_VEL
LIN {X 0,Y 580.258,Z 126.2,A -85,B 0,C 180,E1 -1773.674,E2 -1773.674} C_VEL
LIN {X 0,Y 580.241,Z 126.212,A -85,B 0,C 180,E1 -1776.441,E2 -1776.441} C_VEL
LIN {X 0,Y 580.243,Z 126.202,A -85,B 0,C 180,E1 -1779.436,E2 -1779.436} C_VEL
LIN {X 0,Y 580.237,Z 126.211,A -85,B 0,C 180,E1 -1782.374,E2 -1782.374} C_VEL
LIN {X 0,Y 580.263,Z 126.199,A -85,B 0,C 180,E1 -1785.266,E2 -1785.266} C_VEL
LIN {X 0,Y 580.285,Z 126.207,A -85,B 0,C 180,E1 -1788.119,E2 -1788.119} C_VEL
LIN {X 0,Y 580.238,Z 126.202,A -85,B 0,C 180,E1 -1790.941,E2 -1790.941} C_VEL
LIN {X 0,Y 580.263,Z 126.205,A -85,B 0,C 180,E1 -1793.742,E2 -1793.742} C_VEL
LIN {X 0,Y 580.258,Z 126.208,A -85,B 0,C 180,E1 -1795.833,E2 -1795.833} C_VEL
LIN {X 0,Y 580.341,Z 126.199,A -85,B 0,C 180,E1 -1797.918,E2 -1797.918} C_VEL
LIN {X 0,Y 580.352,Z 126.195,A -85,B 0,C 180,E1 -1800,E2 -1800} C_VEL
LIN {X 0,Y 580.302,Z 126.194,A -85,B 0,C 180,E1 -1802.777,E2 -1802.777} C_VEL
LIN {X 0,Y 580.304,Z 126.202,A -85,B 0,C 180,E1 -1805.56,E2 -1805.56} C_VEL
LIN {X 0,Y 580.296,Z 126.196,A -85,B 0,C 180,E1 -1808.357,E2 -1808.357} C_VEL
LIN {X 0,Y 580.308,Z 126.198,A -85,B 0,C 180,E1 -1811.191,E2 -1811.191} C_VEL
LIN {X 0,Y 580.274,Z 126.198,A -85,B 0,C 180,E1 -1814.32,E2 -1814.32} C_VEL
LIN {X 0,Y 580.256,Z 126.203,A -85,B 0,C 180,E1 -1816.899,E2 -1816.899} C_VEL
LIN {X 0,Y 580.274,Z 126.201,A -85,B 0,C 180,E1 -1819.824,E2 -1819.824} C_VEL
LIN {X 0,Y 580.233,Z 126.203,A -85,B 0,C 180,E1 -1822.055,E2 -1822.055} C_VEL
LIN {X 0,Y 580.278,Z 126.205,A -85,B 0,C 180,E1 -1825.081,E2 -1825.081} C_VEL
LIN {X 0,Y 580.245,Z 126.202,A -85,B 0,C 180,E1 -1827.848,E2 -1827.848} C_VEL
LIN {X 0,Y 580.261,Z 126.204,A -85,B 0,C 180,E1 -1830.689,E2 -1830.689} C_VEL
LIN {X 0,Y 580.282,Z 126.202,A -85,B 0,C 180,E1 -1833.312,E2 -1833.312} C_VEL
LIN {X 0,Y 580.23,Z 126.204,A -85,B 0,C 180,E1 -1835.753,E2 -1835.753} C_VEL
LIN {X 0,Y 580.284,Z 126.197,A -85,B 0,C 180,E1 -1838.147,E2 -1838.147} C_VEL
LIN {X 0,Y 580.296,Z 126.205,A -85,B 0,C 180,E1 -1840.844,E2 -1840.844} C_VEL
LIN {X 0,Y 580.24,Z 126.202,A -85,B 0,C 180,E1 -1843.662,E2 -1843.662} C_VEL
LIN {X 0,Y 580.238,Z 126.212,A -85,B 0,C 180,E1 -1846.614,E2 -1846.614} C_VEL
LIN {X 0,Y 580.293,Z 126.198,A -85,B 0,C 180,E1 -1849.156,E2 -1849.156} C_VEL
LIN {X 0,Y 580.281,Z 126.199,A -85,B 0,C 180,E1 -1851.929,E2 -1851.929} C_VEL
LIN {X 0,Y 580.232,Z 126.213,A -85,B 0,C 180,E1 -1854.451,E2 -1854.451} C_VEL
LIN {X 0,Y 580.286,Z 126.198,A -85,B 0,C 180,E1 -1856.974,E2 -1856.974} C_VEL
LIN {X 0,Y 580.282,Z 126.197,A -85,B 0,C 180,E1 -1859.424,E2 -1859.424} C_VEL
LIN {X 0,Y 580.249,Z 126.209,A -85,B 0,C 180,E1 -1862.151,E2 -1862.151} C_VEL
LIN {X 0,Y 580.283,Z 126.2,A -85,B 0,C 180,E1 -1864.919,E2 -1864.919} C_VEL
LIN {X 0,Y 580.286,Z 126.233,A -85,B 0,C 180,E1 -1866.699,E2 -1866.699} C_VEL
LIN {X 0,Y 580.899,Z 131.051,A -85,B 0,C 180,E1 -1867.41,E2 -1867.41} C_VEL
LIN {X 0,Y 580.78,Z 151.919,A -85,B 0,C 180,E1 -1870.359,E2 -1870.359} C_VEL
LIN {X 0,Y 580.562,Z 174.061,A -85,B 0,C 180,E1 -1873.472,E2 -1873.472} C_VEL
LIN {X 0,Y 580.385,Z 194.611,A -85,B 0,C 180,E1 -1876.319,E2 -1876.319} C_VEL
LIN {X 0,Y 580.936,Z 200.489,A -85,B 0,C 180,E1 -1876.422,E2 -1876.422} C_VEL
LIN {X 0,Y 580.806,Z 302.935,A -85,B 0,C 180,E1 -1877.708,E2 -1877.708} C_VEL
LIN {X 0,Y 580.727,Z 316.211,A -85,B 0,C 180,E1 -1878.017,E2 -1878.017} C_VEL
LIN {X 0,Y 580.648,Z 328.369,A -85,B 0,C 180,E1 -1878.436,E2 -1878.436} C_VEL
LIN {X 0,Y 580.579,Z 340.624,A -85,B 0,C 180,E1 -1879.009,E2 -1879.009} C_VEL
LIN {X 0,Y 580.441,Z 352.198,A -85,B 0,C 180,E1 -1879.712,E2 -1879.712} C_VEL
LIN {X 0,Y 580.345,Z 362.598,A -85,B 0,C 180,E1 -1880.503,E2 -1880.503} C_VEL
LIN {X 0,Y 580.271,Z 371.111,A -85,B 0,C 180,E1 -1881.292,E2 -1881.292} C_VEL
LIN {X 0,Y 580.222,Z 378.959,A -85,B 0,C 180,E1 -1882.168,E2 -1882.168} C_VEL
LIN {X 0,Y 580.154,Z 386.651,A -85,B 0,C 180,E1 -1883.222,E2 -1883.222} C_VEL
LIN {X 0,Y 580.139,Z 393.679,A -85,B 0,C 180,E1 -1884.438,E2 -1884.438} C_VEL
LIN {X 0,Y 580.108,Z 398.371,A -85,B 0,C 180,E1 -1885.483,E2 -1885.483} C_VEL
LIN {X 0,Y 580.123,Z 401.957,A -85,B 0,C 180,E1 -1886.527,E2 -1886.527} C_VEL
LIN {X 0,Y 580.043,Z 403.808,A -85,B 0,C 180,E1 -1887.222,E2 -1887.222} C_VEL
LIN {X 0,Y 580.04,Z 405.198,A -85,B 0,C 180,E1 -1887.917,E2 -1887.917} C_VEL
LIN {X 0,Y 580.04,Z 406.785,A -85,B 0,C 180,E1 -1889.306,E2 -1889.306} C_VEL
LIN {X 0,Y 580.037,Z 407,A -85,B 0,C 180,E1 -1890,E2 -1890} C_VEL
LIN {X 0,Y 580.047,Z 406.186,A -85,B 0,C 180,E1 -1891.388,E2 -1891.388} C_VEL
LIN {X 0,Y 580.04,Z 405.2,A -85,B 0,C 180,E1 -1892.083,E2 -1892.083} C_VEL
LIN {X 0,Y 580.043,Z 403.81,A -85,B 0,C 180,E1 -1892.778,E2 -1892.778} C_VEL
LIN {X 0,Y 580.11,Z 400.896,A -85,B 0,C 180,E1 -1893.82,E2 -1893.82} C_VEL
LIN {X 0,Y 580.053,Z 396.949,A -85,B 0,C 180,E1 -1894.865,E2 -1894.865} C_VEL
LIN {X 0,Y 580.139,Z 390.877,A -85,B 0,C 180,E1 -1896.085,E2 -1896.085} C_VEL
LIN {X 0,Y 580.184,Z 384.238,A -85,B 0,C 180,E1 -1897.132,E2 -1897.132} C_VEL
LIN {X 0,Y 580.25,Z 375.991,A -85,B 0,C 180,E1 -1898.182,E2 -1898.182} C_VEL
LIN {X 0,Y 580.308,Z 367.539,A -85,B 0,C 180,E1 -1899.058,E2 -1899.058} C_VEL
LIN {X 0,Y 580.422,Z 357.099,A -85,B 0,C 180,E1 -1899.936,E2 -1899.936} C_VEL
LIN {X 0,Y 580.506,Z 346.755,A -85,B 0,C 180,E1 -1900.639,E2 -1900.639} C_VEL
LIN {X 0,Y 580.596,Z 335.248,A -85,B 0,C 180,E1 -1901.264,E2 -1901.264} C_VEL
LIN {X 0,Y 580.683,Z 322.472,A -85,B 0,C 180,E1 -1901.785,E2 -1901.785} C_VEL
LIN {X 0,Y 580.778,Z 309.434,A -85,B 0,C 180,E1 -1902.159,E2 -1902.159} C_VEL
LIN {X 0,Y 580.858,Z 297.086,A -85,B 0,C 180,E1 -1902.379,E2 -1902.379} C_VEL
LIN {X 0,Y 580.793,Z 197.381,A -85,B 0,C 180,E1 -1903.621,E2 -1903.621} C_VEL
LIN {X 0,Y 580.387,Z 194.613,A -85,B 0,C 180,E1 -1903.68,E2 -1903.68} C_VEL
LIN {X 0,Y 580.565,Z 172.769,A -85,B 0,C 180,E1 -1906.709,E2 -1906.709} C_VEL
LIN {X 0,Y 580.783,Z 150.762,A -85,B 0,C 180,E1 -1909.805,E2 -1909.805} C_VEL
LIN {X 0,Y 580.899,Z 130.981,A -85,B 0,C 180,E1 -1912.59,E2 -1912.59} C_VEL
LIN {X 0,Y 580.277,Z 126.206,A -85,B 0,C 180,E1 -1913.301,E2 -1913.301} C_VEL
LIN {X 0,Y 580.264,Z 126.209,A -85,B 0,C 180,E1 -1915.85,E2 -1915.85} C_VEL
LIN {X 0,Y 580.279,Z 126.2,A -85,B 0,C 180,E1 -1918.977,E2 -1918.977} C_VEL
LIN {X 0,Y 580.268,Z 126.207,A -85,B 0,C 180,E1 -1921.386,E2 -1921.386} C_VEL
LIN {X 0,Y 580.274,Z 126.202,A -85,B 0,C 180,E1 -1923.858,E2 -1923.858} C_VEL
LIN {X 0,Y 580.277,Z 126.201,A -85,B 0,C 180,E1 -1926.931,E2 -1926.931} C_VEL
LIN {X 0,Y 580.269,Z 126.2,A -85,B 0,C 180,E1 -1929.935,E2 -1929.935} C_VEL
LIN {X 0,Y 580.249,Z 126.204,A -85,B 0,C 180,E1 -1932.709,E2 -1932.709} C_VEL
LIN {X 0,Y 580.252,Z 126.203,A -85,B 0,C 180,E1 -1935.611,E2 -1935.611} C_VEL
LIN {X 0,Y 580.238,Z 126.203,A -85,B 0,C 180,E1 -1938.227,E2 -1938.227} C_VEL
LIN {X 0,Y 580.242,Z 126.211,A -85,B 0,C 180,E1 -1940.962,E2 -1940.962} C_VEL
LIN {X 0,Y 580.229,Z 126.204,A -85,B 0,C 180,E1 -1943.593,E2 -1943.593} C_VEL
LIN {X 0,Y 580.238,Z 126.203,A -85,B 0,C 180,E1 -1946.14,E2 -1946.14} C_VEL
LIN {X 0,Y 580.24,Z 126.212,A -85,B 0,C 180,E1 -1948.612,E2 -1948.612} C_VEL
LIN {X 0,Y 580.244,Z 126.205,A -85,B 0,C 180,E1 -1951.021,E2 -1951.021} C_VEL
LIN {X 0,Y 580.251,Z 126.2,A -85,B 0,C 180,E1 -1953.675,E2 -1953.675} C_VEL
LIN {X 0,Y 580.242,Z 126.211,A -85,B 0,C 180,E1 -1956.44,E2 -1956.44} C_VEL
LIN {X 0,Y 580.245,Z 126.202,A -85,B 0,C 180,E1 -1959.436,E2 -1959.436} C_VEL
LIN {X 0,Y 580.239,Z 126.21,A -85,B 0,C 180,E1 -1962.373,E2 -1962.373} C_VEL
LIN {X 0,Y 580.269,Z 126.199,A -85,B 0,C 180,E1 -1965.265,E2 -1965.265} C_VEL
LIN {X 0,Y 580.293,Z 126.204,A -85,B 0,C 180,E1 -1968.118,E2 -1968.118} C_VEL
LIN {X 0,Y 580.258,Z 126.2,A -85,B 0,C 180,E1 -1970.94,E2 -1970.94} C_VEL
LIN {X 0,Y 580.275,Z 126.206,A -85,B 0,C 180,E1 -1973.742,E2 -1973.742} C_VEL
LIN {X 0,Y 580.264,Z 126.207,A -85,B 0,C 180,E1 -1975.832,E2 -1975.832} C_VEL
LIN {X 0,Y 580.343,Z 126.196,A -85,B 0,C 180,E1 -1977.918,E2 -1977.918} C_VEL
LIN {X 0,Y 580.353,Z 126.192,A -85,B 0,C 180,E1 -1980,E2 -1980} C_VEL
LIN {X 0,Y 580.318,Z 126.193,A -85,B 0,C 180,E1 -1982.776,E2 -1982.776} C_VEL
LIN {X 0,Y 580.318,Z 126.2,A -85,B 0,C 180,E1 -1985.559,E2 -1985.559} C_VEL
LIN {X 0,Y 580.306,Z 126.194,A -85,B 0,C 180,E1 -1988.356,E2 -1988.356} C_VEL
LIN {X 0,Y 580.304,Z 126.202,A -85,B 0,C 180,E1 -1991.191,E2 -1991.191} C_VEL
LIN {X 0,Y 580.309,Z 126.193,A -85,B 0,C 180,E1 -1994.017,E2 -1994.017} C_VEL
LIN {X 0,Y 580.292,Z 126.203,A -85,B 0,C 180,E1 -1996.906,E2 -1996.906} C_VEL
LIN {X 0,Y 580.283,Z 126.198,A -85,B 0,C 180,E1 -1999.823,E2 -1999.823} C_VEL
LIN {X 0,Y 580.286,Z 126.201,A -85,B 0,C 180,E1 -2001.294,E2 -2001.294} C_VEL
LIN {X 0,Y 579.575,Z 126.287,A -85,B 0,C 180,E1 -2001.874,E2 -2001.874} C_VEL
LIN {X 0,Y 576.692,Z 126.652,A -85,B 0,C 180,E1 -2002.813,E2 -2002.813} C_VEL
LIN {X 0,Y 574.295,Z 126.946,A -85,B 0,C 180,E1 -2003.57,E2 -2003.57} C_VEL
LIN {X 0,Y 573.287,Z 127.07,A -85,B 0,C 180,E1 -2004.153,E2 -2004.153} C_VEL
LIN {X 0,Y 573.215,Z 127.08,A -85,B 0,C 180,E1 -2004.351,E2 -2004.351} C_VEL
LIN {X 0,Y 573.249,Z 127.08,A -85,B 0,C 180,E1 -2006.976,E2 -2006.976} C_VEL
LIN {X 0,Y 573.241,Z 127.075,A -85,B 0,C 180,E1 -2009.486,E2 -2009.486} C_VEL
LIN {X 0,Y 573.252,Z 127.082,A -85,B 0,C 180,E1 -2012.645,E2 -2012.645} C_VEL
LIN {X 0,Y 573.206,Z 127.08,A -85,B 0,C 180,E1 -2015.187,E2 -2015.187} C_VEL
LIN {X 0,Y 573.234,Z 127.078,A -85,B 0,C 180,E1 -2017.807,E2 -2017.807} C_VEL
LIN {X 0,Y 573.244,Z 127.082,A -85,B 0,C 180,E1 -2020.525,E2 -2020.525} C_VEL
LIN {X 0,Y 573.24,Z 127.076,A -85,B 0,C 180,E1 -2023.358,E2 -2023.358} C_VEL
LIN {X 0,Y 573.243,Z 127.082,A -85,B 0,C 180,E1 -2026.331,E2 -2026.331} C_VEL
LIN {X 0,Y 573.273,Z 127.074,A -85,B 0,C 180,E1 -2029.477,E2 -2029.477} C_VEL
LIN {X 0,Y 573.272,Z 127.134,A -85,B 0,C 180,E1 -2030.962,E2 -2030.962} C_VEL
LIN {X 0,Y 573.444,Z 134.008,A -85,B 0,C 180,E1 -2032.208,E2 -2032.208} C_VEL
LIN {X 0,Y 573.309,Z 149.825,A -85,B 0,C 180,E1 -2035.05,E2 -2035.05} C_VEL
LIN {X 0,Y 573.248,Z 156.401,A -85,B 0,C 180,E1 -2036.225,E2 -2036.225} C_VEL
LIN {X 0,Y 574.052,Z 161.59,A -85,B 0,C 180,E1 -2036.315,E2 -2036.315} C_VEL
LIN {X 0,Y 573.86,Z 263.184,A -85,B 0,C 180,E1 -2037.607,E2 -2037.607} C_VEL
LIN {X 0,Y 573.787,Z 276.589,A -85,B 0,C 180,E1 -2037.926,E2 -2037.926} C_VEL
LIN {X 0,Y 573.678,Z 289.066,A -85,B 0,C 180,E1 -2038.366,E2 -2038.366} C_VEL
LIN {X 0,Y 573.542,Z 300.728,A -85,B 0,C 180,E1 -2038.923,E2 -2038.923} C_VEL
LIN {X 0,Y 573.427,Z 312.213,A -85,B 0,C 180,E1 -2039.631,E2 -2039.631} C_VEL
LIN {X 0,Y 573.363,Z 323.306,A -85,B 0,C 180,E1 -2040.49,E2 -2040.49} C_VEL
LIN {X 0,Y 573.224,Z 333.04,A -85,B 0,C 180,E1 -2041.435,E2 -2041.435} C_VEL
LIN {X 0,Y 573.147,Z 341.349,A -85,B 0,C 180,E1 -2042.426,E2 -2042.426} C_VEL
LIN {X 0,Y 573.071,Z 348.901,A -85,B 0,C 180,E1 -2043.54,E2 -2043.54} C_VEL
LIN {X 0,Y 573.019,Z 354.503,A -85,B 0,C 180,E1 -2044.579,E2 -2044.579} C_VEL
LIN {X 0,Y 572.987,Z 359.375,A -85,B 0,C 180,E1 -2045.739,E2 -2045.739} C_VEL
LIN {X 0,Y 572.976,Z 363.013,A -85,B 0,C 180,E1 -2046.915,E2 -2046.915} C_VEL
LIN {X 0,Y 572.942,Z 364.676,A -85,B 0,C 180,E1 -2047.65,E2 -2047.65} C_VEL
LIN {X 0,Y 572.961,Z 366.346,A -85,B 0,C 180,E1 -2048.783,E2 -2048.783} C_VEL
LIN {X 0,Y 572.947,Z 366.977,A -85,B 0,C 180,E1 -2049.912,E2 -2049.912} C_VEL
LIN {X 0,Y 572.963,Z 366.739,A -85,B 0,C 180,E1 -2050.818,E2 -2050.818} C_VEL
LIN {X 0,Y 572.943,Z 365.216,A -85,B 0,C 180,E1 -2052.142,E2 -2052.142} C_VEL
LIN {X 0,Y 572.938,Z 363.215,A -85,B 0,C 180,E1 -2053.095,E2 -2053.095} C_VEL
LIN {X 0,Y 572.987,Z 359.396,A -85,B 0,C 180,E1 -2054.345,E2 -2054.345} C_VEL
LIN {X 0,Y 573.028,Z 354.923,A -85,B 0,C 180,E1 -2055.42,E2 -2055.42} C_VEL
LIN {X 0,Y 573.08,Z 349.043,A -85,B 0,C 180,E1 -2056.526,E2 -2056.526} C_VEL
LIN {X 0,Y 573.115,Z 341.781,A -85,B 0,C 180,E1 -2057.608,E2 -2057.608} C_VEL
LIN {X 0,Y 573.206,Z 334.395,A -85,B 0,C 180,E1 -2058.508,E2 -2058.508} C_VEL
LIN {X 0,Y 573.277,Z 325.487,A -85,B 0,C 180,E1 -2059.404,E2 -2059.404} C_VEL
LIN {X 0,Y 573.393,Z 315.719,A -85,B 0,C 180,E1 -2060.209,E2 -2060.209} C_VEL
LIN {X 0,Y 573.545,Z 305.018,A -85,B 0,C 180,E1 -2060.923,E2 -2060.923} C_VEL
LIN {X 0,Y 573.665,Z 293.091,A -85,B 0,C 180,E1 -2061.546,E2 -2061.546} C_VEL
LIN {X 0,Y 573.711,Z 280.757,A -85,B 0,C 180,E1 -2062.034,E2 -2062.034} C_VEL
LIN {X 0,Y 573.797,Z 267.968,A -85,B 0,C 180,E1 -2062.39,E2 -2062.39} C_VEL
LIN {X 0,Y 573.86,Z 254.367,A -85,B 0,C 180,E1 -2062.612,E2 -2062.612} C_VEL
LIN {X 0,Y 573.99,Z 161.06,A -85,B 0,C 180,E1 -2063.784,E2 -2063.784} C_VEL
LIN {X 0,Y 573.206,Z 156.29,A -85,B 0,C 180,E1 -2063.886,E2 -2063.886} C_VEL
LIN {X 0,Y 573.36,Z 141.78,A -85,B 0,C 180,E1 -2066.486,E2 -2066.486} C_VEL
LIN {X 0,Y 573.36,Z 128.204,A -85,B 0,C 180,E1 -2068.947,E2 -2068.947} C_VEL
LIN {X 0,Y 573.188,Z 127.086,A -85,B 0,C 180,E1 -2069.21,E2 -2069.21} C_VEL
LIN {X 0,Y 573.183,Z 127.084,A -85,B 0,C 180,E1 -2070.703,E2 -2070.703} C_VEL
LIN {X 0,Y 573.265,Z 127.073,A -85,B 0,C 180,E1 -2072.811,E2 -2072.811} C_VEL
LIN {X 0,Y 573.262,Z 127.076,A -85,B 0,C 180,E1 -2075.629,E2 -2075.629} C_VEL
LIN {X 0,Y 573.228,Z 127.077,A -85,B 0,C 180,E1 -2078.461,E2 -2078.461} C_VEL
LIN {X 0,Y 573.231,Z 127.078,A -85,B 0,C 180,E1 -2081.313,E2 -2081.313} C_VEL
LIN {X 0,Y 573.231,Z 127.076,A -85,B 0,C 180,E1 -2084.406,E2 -2084.406} C_VEL
LIN {X 0,Y 573.187,Z 127.083,A -85,B 0,C 180,E1 -2087.114,E2 -2087.114} C_VEL
LIN {X 0,Y 573.184,Z 127.084,A -85,B 0,C 180,E1 -2090.079,E2 -2090.079} C_VEL
LIN {X 0,Y 573.188,Z 127.081,A -85,B 0,C 180,E1 -2092.34,E2 -2092.34} C_VEL
LIN {X 0,Y 573.197,Z 127.089,A -85,B 0,C 180,E1 -2095.413,E2 -2095.413} C_VEL
LIN {X 0,Y 573.189,Z 127.082,A -85,B 0,C 180,E1 -2098.018,E2 -2098.018} C_VEL
LIN {X 0,Y 573.197,Z 127.083,A -85,B 0,C 180,E1 -2100.878,E2 -2100.878} C_VEL
LIN {X 0,Y 573.212,Z 127.083,A -85,B 0,C 180,E1 -2103.517,E2 -2103.517} C_VEL
LIN {X 0,Y 573.174,Z 127.083,A -85,B 0,C 180,E1 -2106.055,E2 -2106.055} C_VEL
LIN {X 0,Y 573.214,Z 127.081,A -85,B 0,C 180,E1 -2108.704,E2 -2108.704} C_VEL
LIN {X 0,Y 573.188,Z 127.083,A -85,B 0,C 180,E1 -2111.589,E2 -2111.589} C_VEL
LIN {X 0,Y 573.206,Z 127.083,A -85,B 0,C 180,E1 -2114.674,E2 -2114.674} C_VEL
LIN {X 0,Y 573.2,Z 127.08,A -85,B 0,C 180,E1 -2117.597,E2 -2117.597} C_VEL
LIN {X 0,Y 573.229,Z 127.081,A -85,B 0,C 180,E1 -2120.571,E2 -2120.571} C_VEL
LIN {X 0,Y 573.226,Z 127.081,A -85,B 0,C 180,E1 -2123.076,E2 -2123.076} C_VEL
LIN {X 0,Y 573.231,Z 127.075,A -85,B 0,C 180,E1 -2125.669,E2 -2125.669} C_VEL
LIN {X 0,Y 573.215,Z 127.08,A -85,B 0,C 180,E1 -2128.183,E2 -2128.183} C_VEL
LIN {X 0,Y 573.215,Z 127.086,A -85,B 0,C 180,E1 -2130.632,E2 -2130.632} C_VEL
LIN {X 0,Y 573.201,Z 127.079,A -85,B 0,C 180,E1 -2133.516,E2 -2133.516} C_VEL
LIN {X 0,Y 573.192,Z 127.085,A -85,B 0,C 180,E1 -2136.133,E2 -2136.133} C_VEL
LIN {X 0,Y 573.218,Z 127.077,A -85,B 0,C 180,E1 -2139.173,E2 -2139.173} C_VEL
LIN {X 0,Y 573.198,Z 127.087,A -85,B 0,C 180,E1 -2142.15,E2 -2142.15} C_VEL
LIN {X 0,Y 573.21,Z 127.078,A -85,B 0,C 180,E1 -2145.08,E2 -2145.08} C_VEL
LIN {X 0,Y 573.227,Z 127.083,A -85,B 0,C 180,E1 -2147.97,E2 -2147.97} C_VEL
LIN {X 0,Y 573.204,Z 127.088,A -85,B 0,C 180,E1 -2150.116,E2 -2150.116} C_VEL
LIN {X 0,Y 573.225,Z 127.076,A -85,B 0,C 180,E1 -2152.958,E2 -2152.958} C_VEL
LIN {X 0,Y 573.275,Z 127.07,A -85,B 0,C 180,E1 -2155.077,E2 -2155.077} C_VEL
LIN {X 0,Y 573.31,Z 127.076,A -85,B 0,C 180,E1 -2157.893,E2 -2157.893} C_VEL
LIN {X 0,Y 573.32,Z 127.071,A -85,B 0,C 180,E1 -2160,E2 -2160} C_VEL
LIN {X 0,Y 573.271,Z 127.07,A -85,B 0,C 180,E1 -2162.811,E2 -2162.811} C_VEL
LIN {X 0,Y 573.272,Z 127.079,A -85,B 0,C 180,E1 -2165.629,E2 -2165.629} C_VEL
LIN {X 0,Y 573.237,Z 127.075,A -85,B 0,C 180,E1 -2168.461,E2 -2168.461} C_VEL
LIN {X 0,Y 573.278,Z 127.075,A -85,B 0,C 180,E1 -2171.312,E2 -2171.312} C_VEL
LIN {X 0,Y 573.232,Z 127.075,A -85,B 0,C 180,E1 -2174.402,E2 -2174.402} C_VEL
LIN {X 0,Y 573.198,Z 127.084,A -85,B 0,C 180,E1 -2177.114,E2 -2177.114} C_VEL
LIN {X 0,Y 573.271,Z 127.08,A -85,B 0,C 180,E1 -2179.33,E2 -2179.33} C_VEL
LIN {X 0,Y 573.2,Z 127.079,A -85,B 0,C 180,E1 -2182.34,E2 -2182.34} C_VEL
LIN {X 0,Y 573.226,Z 127.082,A -85,B 0,C 180,E1 -2185.412,E2 -2185.412} C_VEL
LIN {X 0,Y 573.2,Z 127.079,A -85,B 0,C 180,E1 -2188.018,E2 -2188.018} C_VEL
LIN {X 0,Y 573.216,Z 127.084,A -85,B 0,C 180,E1 -2190.879,E2 -2190.879} C_VEL
LIN {X 0,Y 573.247,Z 127.076,A -85,B 0,C 180,E1 -2193.521,E2 -2193.521} C_VEL
LIN {X 0,Y 573.192,Z 127.08,A -85,B 0,C 180,E1 -2196.054,E2 -2196.054} C_VEL
LIN {X 0,Y 573.236,Z 127.082,A -85,B 0,C 180,E1 -2198.702,E2 -2198.702} C_VEL
LIN {X 0,Y 573.217,Z 127.078,A -85,B 0,C 180,E1 -2201.459,E2 -2201.459} C_VEL
LIN {X 0,Y 573.221,Z 127.08,A -85,B 0,C 180,E1 -2204.335,E2 -2204.335} C_VEL
LIN {X 0,Y 573.219,Z 127.078,A -85,B 0,C 180,E1 -2207.361,E2 -2207.361} C_VEL
LIN {X 0,Y 573.233,Z 127.082,A -85,B 0,C 180,E1 -2210.391,E2 -2210.391} C_VEL
LIN {X 0,Y 573.233,Z 127.077,A -85,B 0,C 180,E1 -2213.076,E2 -2213.076} C_VEL
LIN {X 0,Y 573.251,Z 127.073,A -85,B 0,C 180,E1 -2215.67,E2 -2215.67} C_VEL
LIN {X 0,Y 573.229,Z 127.082,A -85,B 0,C 180,E1 -2218.183,E2 -2218.183} C_VEL
LIN {X 0,Y 573.242,Z 127.08,A -85,B 0,C 180,E1 -2220.632,E2 -2220.632} C_VEL
LIN {X 0,Y 573.214,Z 127.08,A -85,B 0,C 180,E1 -2223.513,E2 -2223.513} C_VEL
LIN {X 0,Y 573.241,Z 127.123,A -85,B 0,C 180,E1 -2226.558,E2 -2226.558} C_VEL
LIN {X 0,Y 573.96,Z 132.141,A -85,B 0,C 180,E1 -2227.312,E2 -2227.312} C_VEL
LIN {X 0,Y 573.82,Z 151.864,A -85,B 0,C 180,E1 -2230.131,E2 -2230.131} C_VEL
LIN {X 0,Y 573.589,Z 172.295,A -85,B 0,C 180,E1 -2233.015,E2 -2233.015} C_VEL
LIN {X 0,Y 573.408,Z 193.478,A -85,B 0,C 180,E1 -2235.991,E2 -2235.991} C_VEL
LIN {X 0,Y 573.389,Z 194.611,A -85,B 0,C 180,E1 -2236.149,E2 -2236.149} C_VEL
LIN {X 0,Y 574.049,Z 200.489,A -85,B 0,C 180,E1 -2236.256,E2 -2236.256} C_VEL
LIN {X 0,Y 573.883,Z 302.934,A -85,B 0,C 180,E1 -2237.557,E2 -2237.557} C_VEL
LIN {X 0,Y 573.779,Z 316.21,A -85,B 0,C 180,E1 -2237.869,E2 -2237.869} C_VEL
LIN {X 0,Y 573.699,Z 328.371,A -85,B 0,C 180,E1 -2238.294,E2 -2238.294} C_VEL
LIN {X 0,Y 573.586,Z 340.668,A -85,B 0,C 180,E1 -2238.876,E2 -2238.876} C_VEL
LIN {X 0,Y 573.428,Z 352.195,A -85,B 0,C 180,E1 -2239.585,E2 -2239.585} C_VEL
LIN {X 0,Y 573.333,Z 362.6,A -85,B 0,C 180,E1 -2240.385,E2 -2240.385} C_VEL
LIN {X 0,Y 573.241,Z 371.111,A -85,B 0,C 180,E1 -2241.184,E2 -2241.184} C_VEL
LIN {X 0,Y 573.161,Z 378.959,A -85,B 0,C 180,E1 -2242.071,E2 -2242.071} C_VEL
LIN {X 0,Y 573.073,Z 386.954,A -85,B 0,C 180,E1 -2243.185,E2 -2243.185} C_VEL
LIN {X 0,Y 573.071,Z 393.679,A -85,B 0,C 180,E1 -2244.369,E2 -2244.369} C_VEL
LIN {X 0,Y 573.028,Z 398.372,A -85,B 0,C 180,E1 -2245.427,E2 -2245.427} C_VEL
LIN {X 0,Y 573.022,Z 401.957,A -85,B 0,C 180,E1 -2246.484,E2 -2246.484} C_VEL
LIN {X 0,Y 572.959,Z 403.807,A -85,B 0,C 180,E1 -2247.188,E2 -2247.188} C_VEL
LIN {X 0,Y 572.946,Z 406.185,A -85,B 0,C 180,E1 -2248.594,E2 -2248.594} C_VEL
LIN {X 0,Y 572.938,Z 407,A -85,B 0,C 180,E1 -2250,E2 -2250} C_VEL
LIN {X 0,Y 572.946,Z 406.186,A -85,B 0,C 180,E1 -2251.406,E2 -2251.406} C_VEL
LIN {X 0,Y 572.94,Z 405.199,A -85,B 0,C 180,E1 -2252.109,E2 -2252.109} C_VEL
LIN {X 0,Y 572.959,Z 403.81,A -85,B 0,C 180,E1 -2252.812,E2 -2252.812} C_VEL
LIN {X 0,Y 573.015,Z 400.896,A -85,B 0,C 180,E1 -2253.868,E2 -2253.868} C_VEL
LIN {X 0,Y 572.963,Z 396.949,A -85,B 0,C 180,E1 -2254.926,E2 -2254.926} C_VEL
LIN {X 0,Y 573.065,Z 390.877,A -85,B 0,C 180,E1 -2256.16,E2 -2256.16} C_VEL
LIN {X 0,Y 573.119,Z 384.237,A -85,B 0,C 180,E1 -2257.221,E2 -2257.221} C_VEL
LIN {X 0,Y 573.201,Z 375.992,A -85,B 0,C 180,E1 -2258.283,E2 -2258.283} C_VEL
LIN {X 0,Y 573.287,Z 367.54,A -85,B 0,C 180,E1 -2259.17,E2 -2259.17} C_VEL
LIN {X 0,Y 573.427,Z 357.096,A -85,B 0,C 180,E1 -2260.058,E2 -2260.058} C_VEL
